LIN {X 0,Y 369.698,Z 75.747,A -85,B 0,C 180,E1 18351.289,E2 18351.289} C_VEL
LIN {X 0,Y 369.703,Z 75.746,A -85,B 0,C 180,E1 18347.187,E2 18347.187} C_VEL
LIN {X 0,Y 369.706,Z 75.742,A -85,B 0,C 180,E1 18343.18,E2 18343.18} C_VEL
LIN {X 0,Y 369.715,Z 75.74,A -85,B 0,C 180,E1 18339.085,E2 18339.085} C_VEL
LIN {X 0,Y 369.717,Z 75.741,A -85,B 0,C 180,E1 18335.047,E2 18335.047} C_VEL
LIN {X 0,Y 369.727,Z 75.74,A -85,B 0,C 180,E1 18330.868,E2 18330.868} C_VEL
LIN {X 0,Y 369.716,Z 75.743,A -85,B 0,C 180,E1 18326.888,E2 18326.888} C_VEL
LIN {X 0,Y 369.699,Z 75.747,A -85,B 0,C 180,E1 18322.713,E2 18322.713} C_VEL
LIN {X 0,Y 369.713,Z 75.939,A -85,B 0,C 180,E1 18320.54,E2 18320.54} C_VEL
LIN {X 0,Y 371.263,Z 79.57,A -85,B 0,C 180,E1 18319.328,E2 18319.328} C_VEL
LIN {X 0,Y 375.253,Z 88.261,A -85,B 0,C 180,E1 18316.782,E2 18316.782} C_VEL
LIN {X 0,Y 380.2,Z 100.385,A -85,B 0,C 180,E1 18313.761,E2 18313.761} C_VEL
LIN {X 0,Y 384.853,Z 112.745,A -85,B 0,C 180,E1 18311.095,E2 18311.095} C_VEL
LIN {X 0,Y 389.715,Z 127.844,A -85,B 0,C 180,E1 18308.272,E2 18308.272} C_VEL
LIN {X 0,Y 390.35,Z 131.11,A -85,B 0,C 180,E1 18307.748,E2 18307.748} C_VEL
LIN {X 0,Y 385.426,Z 162.448,A -85,B 0,C 180,E1 18304.176,E2 18304.176} C_VEL
LIN {X 0,Y 388.099,Z 187.157,A -85,B 0,C 180,E1 18303.373,E2 18303.373} C_VEL
LIN {X 0,Y 384.621,Z 335.093,A -85,B 0,C 180,E1 18300.587,E2 18300.587} C_VEL
LIN {X 0,Y 383.923,Z 357.134,A -85,B 0,C 180,E1 18300.105,E2 18300.105} C_VEL
LIN {X 0,Y 382.601,Z 375.427,A -85,B 0,C 180,E1 18299.449,E2 18299.449} C_VEL
LIN {X 0,Y 380.899,Z 392.959,A -85,B 0,C 180,E1 18298.539,E2 18298.539} C_VEL
LIN {X 0,Y 378.892,Z 410.258,A -85,B 0,C 180,E1 18297.334,E2 18297.334} C_VEL
LIN {X 0,Y 376.85,Z 426.215,A -85,B 0,C 180,E1 18295.917,E2 18295.917} C_VEL
LIN {X 0,Y 374.801,Z 441.299,A -85,B 0,C 180,E1 18294.258,E2 18294.258} C_VEL
LIN {X 0,Y 372.823,Z 455.891,A -85,B 0,C 180,E1 18292.295,E2 18292.295} C_VEL
LIN {X 0,Y 371.166,Z 468.894,A -85,B 0,C 180,E1 18290.171,E2 18290.171} C_VEL
LIN {X 0,Y 369.836,Z 480.915,A -85,B 0,C 180,E1 18287.789,E2 18287.789} C_VEL
LIN {X 0,Y 368.946,Z 491.438,A -85,B 0,C 180,E1 18285.242,E2 18285.242} C_VEL
LIN {X 0,Y 368.524,Z 500.454,A -85,B 0,C 180,E1 18282.537,E2 18282.537} C_VEL
LIN {X 0,Y 368.497,Z 507.488,A -85,B 0,C 180,E1 18279.844,E2 18279.844} C_VEL
LIN {X 0,Y 368.76,Z 512.975,A -85,B 0,C 180,E1 18277.009,E2 18277.009} C_VEL
LIN {X 0,Y 369.086,Z 516.444,A -85,B 0,C 180,E1 18274.351,E2 18274.351} C_VEL
LIN {X 0,Y 369.324,Z 518.28,A -85,B 0,C 180,E1 18271.708,E2 18271.708} C_VEL
LIN {X 0,Y 369.368,Z 518.495,A -85,B 0,C 180,E1 18269.071,E2 18269.071} C_VEL
LIN {X 0,Y 369.174,Z 517.092,A -85,B 0,C 180,E1 18266.43,E2 18266.43} C_VEL
LIN {X 0,Y 368.867,Z 514.053,A -85,B 0,C 180,E1 18263.777,E2 18263.777} C_VEL
LIN {X 0,Y 368.587,Z 509.317,A -85,B 0,C 180,E1 18261.106,E2 18261.106} C_VEL
LIN {X 0,Y 368.502,Z 502.683,A -85,B 0,C 180,E1 18258.379,E2 18258.379} C_VEL
LIN {X 0,Y 368.771,Z 494.305,A -85,B 0,C 180,E1 18255.717,E2 18255.717} C_VEL
LIN {X 0,Y 369.45,Z 484.245,A -85,B 0,C 180,E1 18253.169,E2 18253.169} C_VEL
LIN {X 0,Y 370.552,Z 472.63,A -85,B 0,C 180,E1 18250.782,E2 18250.782} C_VEL
LIN {X 0,Y 372.025,Z 459.458,A -85,B 0,C 180,E1 18248.562,E2 18248.562} C_VEL
LIN {X 0,Y 373.773,Z 445.023,A -85,B 0,C 180,E1 18246.569,E2 18246.569} C_VEL
LIN {X 0,Y 375.673,Z 429.361,A -85,B 0,C 180,E1 18244.811,E2 18244.811} C_VEL
LIN {X 0,Y 377.468,Z 413.842,A -85,B 0,C 180,E1 18243.408,E2 18243.408} C_VEL
LIN {X 0,Y 379.259,Z 396.749,A -85,B 0,C 180,E1 18242.186,E2 18242.186} C_VEL
LIN {X 0,Y 380.811,Z 379.266,A -85,B 0,C 180,E1 18241.242,E2 18241.242} C_VEL
LIN {X 0,Y 382.074,Z 360.639,A -85,B 0,C 180,E1 18240.542,E2 18240.542} C_VEL
LIN {X 0,Y 382.7,Z 340.596,A -85,B 0,C 180,E1 18240.083,E2 18240.083} C_VEL
LIN {X 0,Y 386.004,Z 174.055,A -85,B 0,C 180,E1 18237.005,E2 18237.005} C_VEL
LIN {X 0,Y 385.322,Z 157.356,A -85,B 0,C 180,E1 18236.581,E2 18236.581} C_VEL
LIN {X 0,Y 388.344,Z 121.359,A -85,B 0,C 180,E1 18234.252,E2 18234.252} C_VEL
LIN {X 0,Y 379.099,Z 97.949,A -85,B 0,C 180,E1 18231.701,E2 18231.701} C_VEL
LIN {X 0,Y 371.121,Z 79.333,A -85,B 0,C 180,E1 18229.442,E2 18229.442} C_VEL
LIN {X 0,Y 369.792,Z 76.095,A -85,B 0,C 180,E1 18228.97,E2 18228.97} C_VEL
LIN {X 0,Y 369.747,Z 75.737,A -85,B 0,C 180,E1 18228.095,E2 18228.095} C_VEL
LIN {X 0,Y 369.744,Z 75.737,A -85,B 0,C 180,E1 18224.005,E2 18224.005} C_VEL
LIN {X 0,Y 369.744,Z 75.744,A -85,B 0,C 180,E1 18219.829,E2 18219.829} C_VEL
LIN {X 0,Y 369.737,Z 75.735,A -85,B 0,C 180,E1 18215.74,E2 18215.74} C_VEL
LIN {X 0,Y 369.733,Z 75.734,A -85,B 0,C 180,E1 18211.591,E2 18211.591} C_VEL
LIN {X 0,Y 369.731,Z 75.733,A -85,B 0,C 180,E1 18207.505,E2 18207.505} C_VEL
LIN {X 0,Y 369.735,Z 75.729,A -85,B 0,C 180,E1 18203.423,E2 18203.423} C_VEL
LIN {X 0,Y 369.74,Z 75.73,A -85,B 0,C 180,E1 18199.311,E2 18199.311} C_VEL
LIN {X 0,Y 369.75,Z 75.733,A -85,B 0,C 180,E1 18195.129,E2 18195.129} C_VEL
LIN {X 0,Y 369.747,Z 75.739,A -85,B 0,C 180,E1 18191.015,E2 18191.015} C_VEL
LIN {X 0,Y 369.749,Z 75.742,A -85,B 0,C 180,E1 18186.833,E2 18186.833} C_VEL
LIN {X 0,Y 369.732,Z 75.743,A -85,B 0,C 180,E1 18182.635,E2 18182.635} C_VEL
LIN {X 0,Y 369.726,Z 75.738,A -85,B 0,C 180,E1 18178.605,E2 18178.605} C_VEL
LIN {X 0,Y 369.719,Z 75.734,A -85,B 0,C 180,E1 18174.568,E2 18174.568} C_VEL
LIN {X 0,Y 369.716,Z 75.732,A -85,B 0,C 180,E1 18170.504,E2 18170.504} C_VEL
LIN {X 0,Y 369.713,Z 75.733,A -85,B 0,C 180,E1 18166.391,E2 18166.391} C_VEL
LIN {X 0,Y 369.715,Z 75.735,A -85,B 0,C 180,E1 18162.368,E2 18162.368} C_VEL
LIN {X 0,Y 369.718,Z 75.729,A -85,B 0,C 180,E1 18158.253,E2 18158.253} C_VEL
LIN {X 0,Y 369.725,Z 75.734,A -85,B 0,C 180,E1 18154.189,E2 18154.189} C_VEL
LIN {X 0,Y 369.727,Z 75.716,A -85,B 0,C 180,E1 18150.159,E2 18150.159} C_VEL
LIN {X 0,Y 369.734,Z 75.739,A -85,B 0,C 180,E1 18146.117,E2 18146.117} C_VEL
LIN {X 0,Y 369.745,Z 75.747,A -85,B 0,C 180,E1 18141.895,E2 18141.895} C_VEL
LIN {X 0,Y 369.732,Z 75.746,A -85,B 0,C 180,E1 18137.811,E2 18137.811} C_VEL
LIN {X 0,Y 369.73,Z 75.854,A -85,B 0,C 180,E1 18133.661,E2 18133.661} C_VEL
LIN {X 0,Y 370.111,Z 77.451,A -85,B 0,C 180,E1 18133.326,E2 18133.326} C_VEL
LIN {X 0,Y 375.188,Z 90.914,A -85,B 0,C 180,E1 18131.164,E2 18131.164} C_VEL
LIN {X 0,Y 380.295,Z 107.557,A -85,B 0,C 180,E1 18128.66,E2 18128.66} C_VEL
LIN {X 0,Y 381.618,Z 113.58,A -85,B 0,C 180,E1 18127.811,E2 18127.811} C_VEL
LIN {X 0,Y 380.63,Z 148.33,A -85,B 0,C 180,E1 18123.749,E2 18123.749} C_VEL
LIN {X 0,Y 379.687,Z 184.035,A -85,B 0,C 180,E1 18119.655,E2 18119.655} C_VEL
LIN {X 0,Y 379.452,Z 200.957,A -85,B 0,C 180,E1 18117.821,E2 18117.821} C_VEL
LIN {X 0,Y 380.058,Z 205.985,A -85,B 0,C 180,E1 18117.673,E2 18117.673} C_VEL
LIN {X 0,Y 378.353,Z 307.859,A -85,B 0,C 180,E1 18115.716,E2 18115.716} C_VEL
LIN {X 0,Y 378.281,Z 322.743,A -85,B 0,C 180,E1 18115.252,E2 18115.252} C_VEL
LIN {X 0,Y 377.861,Z 336.788,A -85,B 0,C 180,E1 18114.545,E2 18114.545} C_VEL
LIN {X 0,Y 377.058,Z 350.975,A -85,B 0,C 180,E1 18113.519,E2 18113.519} C_VEL
LIN {X 0,Y 376.047,Z 363.63,A -85,B 0,C 180,E1 18112.287,E2 18112.287} C_VEL
LIN {X 0,Y 374.946,Z 375.143,A -85,B 0,C 180,E1 18110.836,E2 18110.836} C_VEL
LIN {X 0,Y 373.79,Z 385.284,A -85,B 0,C 180,E1 18109.207,E2 18109.207} C_VEL
LIN {X 0,Y 372.627,Z 394.373,A -85,B 0,C 180,E1 18107.327,E2 18107.327} C_VEL
LIN {X 0,Y 371.679,Z 401.417,A -85,B 0,C 180,E1 18105.444,E2 18105.444} C_VEL
LIN {X 0,Y 370.832,Z 407.525,A -85,B 0,C 180,E1 18103.247,E2 18103.247} C_VEL
LIN {X 0,Y 370.196,Z 411.9,A -85,B 0,C 180,E1 18100.897,E2 18100.897} C_VEL
LIN {X 0,Y 369.808,Z 414.328,A -85,B 0,C 180,E1 18098.551,E2 18098.551} C_VEL
LIN {X 0,Y 369.626,Z 414.959,A -85,B 0,C 180,E1 18096.21,E2 18096.21} C_VEL
LIN {X 0,Y 369.636,Z 413.831,A -85,B 0,C 180,E1 18093.876,E2 18093.876} C_VEL
LIN {X 0,Y 369.858,Z 410.615,A -85,B 0,C 180,E1 18091.393,E2 18091.393} C_VEL
LIN {X 0,Y 370.279,Z 405.57,A -85,B 0,C 180,E1 18089.071,E2 18089.071} C_VEL
LIN {X 0,Y 370.837,Z 399.392,A -85,B 0,C 180,E1 18087.062,E2 18087.062} C_VEL
LIN {X 0,Y 371.6,Z 391.246,A -85,B 0,C 180,E1 18085.06,E2 18085.06} C_VEL
LIN {X 0,Y 372.064,Z 386.159,A -85,B 0,C 180,E1 18084.043,E2 18084.043} C_VEL
LIN {X 0,Y 371.549,Z 381.232,A -85,B 0,C 180,E1 18083.121,E2 18083.121} C_VEL
LIN {X 0,Y 368.041,Z 371.768,A -85,B 0,C 180,E1 18081.5,E2 18081.5} C_VEL
LIN {X 0,Y 366.43,Z 365.291,A -85,B 0,C 180,E1 18080.582,E2 18080.582} C_VEL
LIN {X 0,Y 366.351,Z 361.699,A -85,B 0,C 180,E1 18080.163,E2 18080.163} C_VEL
LIN {X 0,Y 367.154,Z 348.44,A -85,B 0,C 180,E1 18078.93,E2 18078.93} C_VEL
LIN {X 0,Y 367.732,Z 334.792,A -85,B 0,C 180,E1 18077.994,E2 18077.994} C_VEL
LIN {X 0,Y 368,Z 320.348,A -85,B 0,C 180,E1 18077.305,E2 18077.305} C_VEL
LIN {X 0,Y 367.969,Z 303.735,A -85,B 0,C 180,E1 18076.855,E2 18076.855} C_VEL
LIN {X 0,Y 369.693,Z 197.834,A -85,B 0,C 180,E1 18074.79,E2 18074.79} C_VEL
LIN {X 0,Y 370.403,Z 188.265,A -85,B 0,C 180,E1 18074.178,E2 18074.178} C_VEL
LIN {X 0,Y 370.622,Z 185.191,A -85,B 0,C 180,E1 18073.906,E2 18073.906} C_VEL
LIN {X 0,Y 371.261,Z 184.243,A -85,B 0,C 180,E1 18073.653,E2 18073.653} C_VEL
LIN {X 0,Y 372.216,Z 184.586,A -85,B 0,C 180,E1 18073.476,E2 18073.476} C_VEL
LIN {X 0,Y 374.171,Z 186.02,A -85,B 0,C 180,E1 18073.295,E2 18073.295} C_VEL
LIN {X 0,Y 374.868,Z 197.394,A -85,B 0,C 180,E1 18072.973,E2 18072.973} C_VEL
LIN {X 0,Y 371.793,Z 301.218,A -85,B 0,C 180,E1 18070.645,E2 18070.645} C_VEL
LIN {X 0,Y 371.137,Z 317.525,A -85,B 0,C 180,E1 18069.992,E2 18069.992} C_VEL
LIN {X 0,Y 370.215,Z 332.434,A -85,B 0,C 180,E1 18069.114,E2 18069.114} C_VEL
LIN {X 0,Y 369.084,Z 346.795,A -85,B 0,C 180,E1 18067.986,E2 18067.986} C_VEL
LIN {X 0,Y 367.697,Z 361.204,A -85,B 0,C 180,E1 18066.5,E2 18066.5} C_VEL
LIN {X 0,Y 366.448,Z 373.045,A -85,B 0,C 180,E1 18064.941,E2 18064.941} C_VEL
LIN {X 0,Y 365.194,Z 383.994,A -85,B 0,C 180,E1 18063.143,E2 18063.143} C_VEL
LIN {X 0,Y 364.03,Z 393.789,A -85,B 0,C 180,E1 18061.091,E2 18061.091} C_VEL
LIN {X 0,Y 363.098,Z 401.859,A -85,B 0,C 180,E1 18058.915,E2 18058.915} C_VEL
LIN {X 0,Y 362.369,Z 408.627,A -85,B 0,C 180,E1 18056.439,E2 18056.439} C_VEL
LIN {X 0,Y 361.944,Z 413.075,A -85,B 0,C 180,E1 18054.039,E2 18054.039} C_VEL
LIN {X 0,Y 361.762,Z 415.798,A -85,B 0,C 180,E1 18051.547,E2 18051.547} C_VEL
LIN {X 0,Y 361.815,Z 416.609,A -85,B 0,C 180,E1 18048.976,E2 18048.976} C_VEL
LIN {X 0,Y 362.098,Z 415.605,A -85,B 0,C 180,E1 18046.562,E2 18046.562} C_VEL
LIN {X 0,Y 362.68,Z 412.568,A -85,B 0,C 180,E1 18043.983,E2 18043.983} C_VEL
LIN {X 0,Y 363.459,Z 408.133,A -85,B 0,C 180,E1 18041.739,E2 18041.739} C_VEL
LIN {X 0,Y 364.635,Z 401.413,A -85,B 0,C 180,E1 18039.351,E2 18039.351} C_VEL
LIN {X 0,Y 366.023,Z 393.164,A -85,B 0,C 180,E1 18037.196,E2 18037.196} C_VEL
LIN {X 0,Y 367.611,Z 383.402,A -85,B 0,C 180,E1 18035.213,E2 18035.213} C_VEL
LIN {X 0,Y 369.378,Z 371.52,A -85,B 0,C 180,E1 18033.333,E2 18033.333} C_VEL
LIN {X 0,Y 371.018,Z 359.359,A -85,B 0,C 180,E1 18031.817,E2 18031.817} C_VEL
LIN {X 0,Y 372.676,Z 345.086,A -85,B 0,C 180,E1 18030.42,E2 18030.42} C_VEL
LIN {X 0,Y 374.102,Z 329.6,A -85,B 0,C 180,E1 18029.282,E2 18029.282} C_VEL
LIN {X 0,Y 375.148,Z 314.19,A -85,B 0,C 180,E1 18028.461,E2 18028.461} C_VEL
LIN {X 0,Y 375.878,Z 297.331,A -85,B 0,C 180,E1 18027.87,E2 18027.87} C_VEL
LIN {X 0,Y 379.463,Z 207.466,A -85,B 0,C 180,E1 18025.682,E2 18025.682} C_VEL
LIN {X 0,Y 374.321,Z 178.027,A -85,B 0,C 180,E1 18024.332,E2 18024.332} C_VEL
LIN {X 0,Y 373.222,Z 172.209,A -85,B 0,C 180,E1 18024.001,E2 18024.001} C_VEL
LIN {X 0,Y 377.007,Z 145.712,A -85,B 0,C 180,E1 18019.683,E2 18019.683} C_VEL
LIN {X 0,Y 379.418,Z 130.52,A -85,B 0,C 180,E1 18017.167,E2 18017.167} C_VEL
LIN {X 0,Y 376.228,Z 117.259,A -85,B 0,C 180,E1 18014.153,E2 18014.153} C_VEL
LIN {X 0,Y 372.504,Z 104.805,A -85,B 0,C 180,E1 18010.987,E2 18010.987} C_VEL
LIN {X 0,Y 368.787,Z 94.247,A -85,B 0,C 180,E1 18007.948,E2 18007.948} C_VEL
LIN {X 0,Y 365.768,Z 86.709,A -85,B 0,C 180,E1 18005.491,E2 18005.491} C_VEL
LIN {X 0,Y 363.086,Z 80.246,A -85,B 0,C 180,E1 18003.158,E2 18003.158} C_VEL
LIN {X 0,Y 361.785,Z 76.834,A -85,B 0,C 180,E1 18001.742,E2 18001.742} C_VEL
LIN {X 0,Y 361.766,Z 76.732,A -85,B 0,C 180,E1 17997.783,E2 17997.783} C_VEL
LIN {X 0,Y 361.759,Z 76.733,A -85,B 0,C 180,E1 17993.653,E2 17993.653} C_VEL
LIN {X 0,Y 361.757,Z 76.734,A -85,B 0,C 180,E1 17989.49,E2 17989.49} C_VEL
LIN {X 0,Y 361.76,Z 76.732,A -85,B 0,C 180,E1 17985.321,E2 17985.321} C_VEL
LIN {X 0,Y 361.761,Z 76.73,A -85,B 0,C 180,E1 17981.301,E2 17981.301} C_VEL
LIN {X 0,Y 361.767,Z 76.73,A -85,B 0,C 180,E1 17977.236,E2 17977.236} C_VEL
LIN {X 0,Y 361.781,Z 76.729,A -85,B 0,C 180,E1 17973.048,E2 17973.048} C_VEL
LIN {X 0,Y 361.786,Z 76.73,A -85,B 0,C 180,E1 17968.882,E2 17968.882} C_VEL
LIN {X 0,Y 361.764,Z 76.738,A -85,B 0,C 180,E1 17964.715,E2 17964.715} C_VEL
LIN {X 0,Y 361.784,Z 77.027,A -85,B 0,C 180,E1 17962.286,E2 17962.286} C_VEL
LIN {X 0,Y 363.536,Z 80.865,A -85,B 0,C 180,E1 17960.861,E2 17960.861} C_VEL
LIN {X 0,Y 366.269,Z 87.098,A -85,B 0,C 180,E1 17958.861,E2 17958.861} C_VEL
LIN {X 0,Y 369.245,Z 93.448,A -85,B 0,C 180,E1 17956.971,E2 17956.971} C_VEL
LIN {X 0,Y 373.932,Z 105.09,A -85,B 0,C 180,E1 17954.005,E2 17954.005} C_VEL
LIN {X 0,Y 378.636,Z 117.95,A -85,B 0,C 180,E1 17951.185,E2 17951.185} C_VEL
LIN {X 0,Y 383.225,Z 132.648,A -85,B 0,C 180,E1 17948.387,E2 17948.387} C_VEL
LIN {X 0,Y 383.339,Z 133.981,A -85,B 0,C 180,E1 17948.183,E2 17948.183} C_VEL
LIN {X 0,Y 378.588,Z 162.637,A -85,B 0,C 180,E1 17944.852,E2 17944.852} C_VEL
LIN {X 0,Y 381.297,Z 187.979,A -85,B 0,C 180,E1 17943.991,E2 17943.991} C_VEL
LIN {X 0,Y 377.104,Z 352.179,A -85,B 0,C 180,E1 17940.807,E2 17940.807} C_VEL
LIN {X 0,Y 375.864,Z 370.525,A -85,B 0,C 180,E1 17940.195,E2 17940.195} C_VEL
LIN {X 0,Y 374.052,Z 388.976,A -85,B 0,C 180,E1 17939.287,E2 17939.287} C_VEL
LIN {X 0,Y 372.051,Z 406.054,A -85,B 0,C 180,E1 17938.142,E2 17938.142} C_VEL
LIN {X 0,Y 369.904,Z 422.137,A -85,B 0,C 180,E1 17936.76,E2 17936.76} C_VEL
LIN {X 0,Y 367.712,Z 437.614,A -85,B 0,C 180,E1 17935.1,E2 17935.1} C_VEL
LIN {X 0,Y 365.616,Z 452.083,A -85,B 0,C 180,E1 17933.192,E2 17933.192} C_VEL
LIN {X 0,Y 363.675,Z 465.993,A -85,B 0,C 180,E1 17930.942,E2 17930.942} C_VEL
LIN {X 0,Y 362.166,Z 478.323,A -85,B 0,C 180,E1 17928.512,E2 17928.512} C_VEL
LIN {X 0,Y 361.12,Z 489.113,A -85,B 0,C 180,E1 17925.91,E2 17925.91} C_VEL
LIN {X 0,Y 360.586,Z 498.36,A -85,B 0,C 180,E1 17923.144,E2 17923.144} C_VEL
LIN {X 0,Y 360.493,Z 505.612,A -85,B 0,C 180,E1 17920.387,E2 17920.387} C_VEL
LIN {X 0,Y 360.724,Z 511.064,A -85,B 0,C 180,E1 17917.647,E2 17917.647} C_VEL
LIN {X 0,Y 361.07,Z 514.813,A -85,B 0,C 180,E1 17914.926,E2 17914.926} C_VEL
LIN {X 0,Y 361.364,Z 516.927,A -85,B 0,C 180,E1 17912.221,E2 17912.221} C_VEL
LIN {X 0,Y 361.457,Z 517.425,A -85,B 0,C 180,E1 17909.526,E2 17909.526} C_VEL
LIN {X 0,Y 361.286,Z 516.294,A -85,B 0,C 180,E1 17906.828,E2 17906.828} C_VEL
LIN {X 0,Y 360.963,Z 513.519,A -85,B 0,C 180,E1 17904.119,E2 17904.119} C_VEL
LIN {X 0,Y 360.649,Z 509.047,A -85,B 0,C 180,E1 17901.391,E2 17901.391} C_VEL
LIN {X 0,Y 360.519,Z 502.362,A -85,B 0,C 180,E1 17898.483,E2 17898.483} C_VEL
LIN {X 0,Y 360.748,Z 494.584,A -85,B 0,C 180,E1 17895.884,E2 17895.884} C_VEL
LIN {X 0,Y 361.398,Z 484.846,A -85,B 0,C 180,E1 17893.279,E2 17893.279} C_VEL
LIN {X 0,Y 362.492,Z 473.616,A -85,B 0,C 180,E1 17890.84,E2 17890.84} C_VEL
LIN {X 0,Y 363.968,Z 460.882,A -85,B 0,C 180,E1 17888.572,E2 17888.572} C_VEL
LIN {X 0,Y 365.777,Z 446.469,A -85,B 0,C 180,E1 17886.48,E2 17886.48} C_VEL
LIN {X 0,Y 367.66,Z 431.673,A -85,B 0,C 180,E1 17884.727,E2 17884.727} C_VEL
LIN {X 0,Y 369.57,Z 416.07,A -85,B 0,C 180,E1 17883.227,E2 17883.227} C_VEL
LIN {X 0,Y 371.385,Z 399.763,A -85,B 0,C 180,E1 17881.981,E2 17881.981} C_VEL
LIN {X 0,Y 373.104,Z 381.924,A -85,B 0,C 180,E1 17880.942,E2 17880.942} C_VEL
LIN {X 0,Y 374.476,Z 363.631,A -85,B 0,C 180,E1 17880.185,E2 17880.185} C_VEL
LIN {X 0,Y 375.234,Z 345.261,A -85,B 0,C 180,E1 17879.701,E2 17879.701} C_VEL
LIN {X 0,Y 378.813,Z 174.715,A -85,B 0,C 180,E1 17876.489,E2 17876.489} C_VEL
LIN {X 0,Y 378.136,Z 157.313,A -85,B 0,C 180,E1 17876.036,E2 17876.036} C_VEL
LIN {X 0,Y 381.061,Z 123.76,A -85,B 0,C 180,E1 17873.819,E2 17873.819} C_VEL
LIN {X 0,Y 371.694,Z 99.975,A -85,B 0,C 180,E1 17871.147,E2 17871.147} C_VEL
LIN {X 0,Y 362.82,Z 79.739,A -85,B 0,C 180,E1 17868.596,E2 17868.596} C_VEL
LIN {X 0,Y 361.856,Z 77.053,A -85,B 0,C 180,E1 17868.192,E2 17868.192} C_VEL
LIN {X 0,Y 361.8,Z 76.732,A -85,B 0,C 180,E1 17867.172,E2 17867.172} C_VEL
LIN {X 0,Y 361.804,Z 76.729,A -85,B 0,C 180,E1 17862.92,E2 17862.92} C_VEL
LIN {X 0,Y 361.813,Z 76.725,A -85,B 0,C 180,E1 17858.807,E2 17858.807} C_VEL
LIN {X 0,Y 361.81,Z 76.723,A -85,B 0,C 180,E1 17854.565,E2 17854.565} C_VEL
LIN {X 0,Y 361.815,Z 76.727,A -85,B 0,C 180,E1 17850.378,E2 17850.378} C_VEL
LIN {X 0,Y 361.803,Z 76.729,A -85,B 0,C 180,E1 17846.242,E2 17846.242} C_VEL
LIN {X 0,Y 361.797,Z 76.729,A -85,B 0,C 180,E1 17842.076,E2 17842.076} C_VEL
LIN {X 0,Y 361.788,Z 76.728,A -85,B 0,C 180,E1 17837.864,E2 17837.864} C_VEL
LIN {X 0,Y 361.788,Z 76.722,A -85,B 0,C 180,E1 17833.749,E2 17833.749} C_VEL
LIN {X 0,Y 361.794,Z 76.716,A -85,B 0,C 180,E1 17829.544,E2 17829.544} C_VEL
LIN {X 0,Y 361.797,Z 76.724,A -85,B 0,C 180,E1 17825.55,E2 17825.55} C_VEL
LIN {X 0,Y 361.805,Z 76.728,A -85,B 0,C 180,E1 17821.425,E2 17821.425} C_VEL
LIN {X 0,Y 361.806,Z 76.73,A -85,B 0,C 180,E1 17817.307,E2 17817.307} C_VEL
LIN {X 0,Y 361.813,Z 76.728,A -85,B 0,C 180,E1 17813.175,E2 17813.175} C_VEL
LIN {X 0,Y 361.793,Z 76.728,A -85,B 0,C 180,E1 17809.007,E2 17809.007} C_VEL
LIN {X 0,Y 361.785,Z 76.727,A -85,B 0,C 180,E1 17804.942,E2 17804.942} C_VEL
LIN {X 0,Y 361.777,Z 76.731,A -85,B 0,C 180,E1 17800.798,E2 17800.798} C_VEL
LIN {X 0,Y 361.772,Z 76.694,A -85,B 0,C 180,E1 17796.547,E2 17796.547} C_VEL
LIN {X 0,Y 361.775,Z 76.733,A -85,B 0,C 180,E1 17792.512,E2 17792.512} C_VEL
LIN {X 0,Y 361.773,Z 76.716,A -85,B 0,C 180,E1 17788.509,E2 17788.509} C_VEL
LIN {X 0,Y 361.772,Z 76.712,A -85,B 0,C 180,E1 17784.521,E2 17784.521} C_VEL
LIN {X 0,Y 361.778,Z 76.72,A -85,B 0,C 180,E1 17780.448,E2 17780.448} C_VEL
LIN {X 0,Y 361.791,Z 76.718,A -85,B 0,C 180,E1 17776.297,E2 17776.297} C_VEL
LIN {X 0,Y 361.825,Z 76.996,A -85,B 0,C 180,E1 17774.382,E2 17774.382} C_VEL
LIN {X 0,Y 368.457,Z 95.021,A -85,B 0,C 180,E1 17771.381,E2 17771.381} C_VEL
LIN {X 0,Y 373.513,Z 111.76,A -85,B 0,C 180,E1 17768.832,E2 17768.832} C_VEL
LIN {X 0,Y 374.46,Z 116.271,A -85,B 0,C 180,E1 17768.188,E2 17768.188} C_VEL
LIN {X 0,Y 373.374,Z 151.557,A -85,B 0,C 180,E1 17764.032,E2 17764.032} C_VEL
LIN {X 0,Y 372.387,Z 187.837,A -85,B 0,C 180,E1 17759.858,E2 17759.858} C_VEL
LIN {X 0,Y 372.146,Z 201.909,A -85,B 0,C 180,E1 17758.325,E2 17758.325} C_VEL
LIN {X 0,Y 372.787,Z 207.087,A -85,B 0,C 180,E1 17758.168,E2 17758.168} C_VEL
LIN {X 0,Y 370.982,Z 308.241,A -85,B 0,C 180,E1 17756.189,E2 17756.189} C_VEL
LIN {X 0,Y 370.914,Z 323.342,A -85,B 0,C 180,E1 17755.72,E2 17755.72} C_VEL
LIN {X 0,Y 370.457,Z 337.796,A -85,B 0,C 180,E1 17754.984,E2 17754.984} C_VEL
LIN {X 0,Y 369.609,Z 352.011,A -85,B 0,C 180,E1 17753.938,E2 17753.938} C_VEL
LIN {X 0,Y 368.582,Z 364.251,A -85,B 0,C 180,E1 17752.731,E2 17752.731} C_VEL
LIN {X 0,Y 367.455,Z 375.561,A -85,B 0,C 180,E1 17751.299,E2 17751.299} C_VEL
LIN {X 0,Y 366.099,Z 386.791,A -85,B 0,C 180,E1 17749.461,E2 17749.461} C_VEL
LIN {X 0,Y 364.786,Z 396.461,A -85,B 0,C 180,E1 17747.382,E2 17747.382} C_VEL
LIN {X 0,Y 363.658,Z 404.236,A -85,B 0,C 180,E1 17745.14,E2 17745.14} C_VEL
LIN {X 0,Y 362.814,Z 409.801,A -85,B 0,C 180,E1 17742.897,E2 17742.897} C_VEL
LIN {X 0,Y 362.233,Z 413.52,A -85,B 0,C 180,E1 17740.656,E2 17740.656} C_VEL
LIN {X 0,Y 361.855,Z 415.673,A -85,B 0,C 180,E1 17738.26,E2 17738.26} C_VEL
LIN {X 0,Y 361.688,Z 415.965,A -85,B 0,C 180,E1 17735.71,E2 17735.71} C_VEL
LIN {X 0,Y 361.747,Z 414.228,A -85,B 0,C 180,E1 17733.168,E2 17733.168} C_VEL
LIN {X 0,Y 362.019,Z 410.7,A -85,B 0,C 180,E1 17730.79,E2 17730.79} C_VEL
LIN {X 0,Y 362.475,Z 405.614,A -85,B 0,C 180,E1 17728.576,E2 17728.576} C_VEL
LIN {X 0,Y 363.106,Z 399.118,A -85,B 0,C 180,E1 17726.526,E2 17726.526} C_VEL
LIN {X 0,Y 363.944,Z 390.508,A -85,B 0,C 180,E1 17724.481,E2 17724.481} C_VEL
LIN {X 0,Y 364.816,Z 381.152,A -85,B 0,C 180,E1 17722.756,E2 17722.756} C_VEL
LIN {X 0,Y 365.775,Z 369.814,A -85,B 0,C 180,E1 17721.114,E2 17721.114} C_VEL
LIN {X 0,Y 366.351,Z 361.699,A -85,B 0,C 180,E1 17720.163,E2 17720.163} C_VEL
LIN {X 0,Y 365.835,Z 355.352,A -85,B 0,C 180,E1 17719.464,E2 17719.464} C_VEL
LIN {X 0,Y 362.537,Z 344.434,A -85,B 0,C 180,E1 17718.347,E2 17718.347} C_VEL
LIN {X 0,Y 360.593,Z 336.68,A -85,B 0,C 180,E1 17717.72,E2 17717.72} C_VEL
LIN {X 0,Y 360.219,Z 331.508,A -85,B 0,C 180,E1 17717.407,E2 17717.407} C_VEL
LIN {X 0,Y 360.411,Z 316.564,A -85,B 0,C 180,E1 17716.778,E2 17716.778} C_VEL
LIN {X 0,Y 360.589,Z 278.756,A -85,B 0,C 180,E1 17715.965,E2 17715.965} C_VEL
LIN {X 0,Y 362.164,Z 199.347,A -85,B 0,C 180,E1 17714.384,E2 17714.384} C_VEL
LIN {X 0,Y 362.67,Z 196.935,A -85,B 0,C 180,E1 17714.16,E2 17714.16} C_VEL
LIN {X 0,Y 363.659,Z 196.064,A -85,B 0,C 180,E1 17713.876,E2 17713.876} C_VEL
LIN {X 0,Y 365.776,Z 197.599,A -85,B 0,C 180,E1 17713.633,E2 17713.633} C_VEL
LIN {X 0,Y 367.619,Z 197.786,A -85,B 0,C 180,E1 17713.492,E2 17713.492} C_VEL
LIN {X 0,Y 364.392,Z 301.648,A -85,B 0,C 180,E1 17711.113,E2 17711.113} C_VEL
LIN {X 0,Y 363.702,Z 318.046,A -85,B 0,C 180,E1 17710.445,E2 17710.445} C_VEL
LIN {X 0,Y 362.69,Z 333.639,A -85,B 0,C 180,E1 17709.505,E2 17709.505} C_VEL
LIN {X 0,Y 361.488,Z 348.073,A -85,B 0,C 180,E1 17708.337,E2 17708.337} C_VEL
LIN {X 0,Y 360.041,Z 362.488,A -85,B 0,C 180,E1 17706.812,E2 17706.812} C_VEL
LIN {X 0,Y 358.642,Z 375.026,A -85,B 0,C 180,E1 17705.103,E2 17705.103} C_VEL
LIN {X 0,Y 357.319,Z 385.995,A -85,B 0,C 180,E1 17703.222,E2 17703.222} C_VEL
LIN {X 0,Y 356.128,Z 395.608,A -85,B 0,C 180,E1 17701.124,E2 17701.124} C_VEL
LIN {X 0,Y 355.204,Z 403.19,A -85,B 0,C 180,E1 17698.993,E2 17698.993} C_VEL
LIN {X 0,Y 354.484,Z 409.569,A -85,B 0,C 180,E1 17696.606,E2 17696.606} C_VEL
LIN {X 0,Y 354.044,Z 413.975,A -85,B 0,C 180,E1 17694.225,E2 17694.225} C_VEL
LIN {X 0,Y 353.844,Z 416.737,A -85,B 0,C 180,E1 17691.769,E2 17691.769} C_VEL
LIN {X 0,Y 353.877,Z 417.734,A -85,B 0,C 180,E1 17689.22,E2 17689.22} C_VEL
LIN {X 0,Y 354.167,Z 416.947,A -85,B 0,C 180,E1 17686.683,E2 17686.683} C_VEL
LIN {X 0,Y 354.697,Z 414.42,A -85,B 0,C 180,E1 17684.274,E2 17684.274} C_VEL
LIN {X 0,Y 355.553,Z 410.005,A -85,B 0,C 180,E1 17681.796,E2 17681.796} C_VEL
LIN {X 0,Y 356.659,Z 404.042,A -85,B 0,C 180,E1 17679.522,E2 17679.522} C_VEL
LIN {X 0,Y 358.106,Z 396.168,A -85,B 0,C 180,E1 17677.274,E2 17677.274} C_VEL
LIN {X 0,Y 359.759,Z 386.663,A -85,B 0,C 180,E1 17675.204,E2 17675.204} C_VEL
LIN {X 0,Y 361.517,Z 375.933,A -85,B 0,C 180,E1 17673.357,E2 17673.357} C_VEL
LIN {X 0,Y 363.433,Z 362.862,A -85,B 0,C 180,E1 17671.599,E2 17671.599} C_VEL
LIN {X 0,Y 365.04,Z 350.233,A -85,B 0,C 180,E1 17670.264,E2 17670.264} C_VEL
LIN {X 0,Y 366.612,Z 335.35,A -85,B 0,C 180,E1 17669.043,E2 17669.043} C_VEL
LIN {X 0,Y 367.802,Z 320.518,A -85,B 0,C 180,E1 17668.142,E2 17668.142} C_VEL
LIN {X 0,Y 368.713,Z 304.032,A -85,B 0,C 180,E1 17667.447,E2 17667.447} C_VEL
LIN {X 0,Y 372.74,Z 208.847,A -85,B 0,C 180,E1 17665.045,E2 17665.045} C_VEL
LIN {X 0,Y 367.735,Z 179.907,A -85,B 0,C 180,E1 17663.676,E2 17663.676} C_VEL
LIN {X 0,Y 366.264,Z 172.119,A -85,B 0,C 180,E1 17663.233,E2 17663.233} C_VEL
LIN {X 0,Y 370.459,Z 144.692,A -85,B 0,C 180,E1 17658.676,E2 17658.676} C_VEL
LIN {X 0,Y 372.276,Z 133.118,A -85,B 0,C 180,E1 17656.702,E2 17656.702} C_VEL
LIN {X 0,Y 369.147,Z 120.062,A -85,B 0,C 180,E1 17653.63,E2 17653.63} C_VEL
LIN {X 0,Y 365.502,Z 107.842,A -85,B 0,C 180,E1 17650.402,E2 17650.402} C_VEL
LIN {X 0,Y 361.732,Z 96.884,A -85,B 0,C 180,E1 17647.11,E2 17647.11} C_VEL
LIN {X 0,Y 358.264,Z 88.443,A -85,B 0,C 180,E1 17644.161,E2 17644.161} C_VEL
LIN {X 0,Y 356.657,Z 84.754,A -85,B 0,C 180,E1 17642.732,E2 17642.732} C_VEL
LIN {X 0,Y 355.168,Z 81.263,A -85,B 0,C 180,E1 17641.291,E2 17641.291} C_VEL
LIN {X 0,Y 353.84,Z 77.821,A -85,B 0,C 180,E1 17639.677,E2 17639.677} C_VEL
LIN {X 0,Y 353.821,Z 77.723,A -85,B 0,C 180,E1 17635.462,E2 17635.462} C_VEL
LIN {X 0,Y 353.819,Z 77.724,A -85,B 0,C 180,E1 17631.387,E2 17631.387} C_VEL
LIN {X 0,Y 353.822,Z 77.723,A -85,B 0,C 180,E1 17627.267,E2 17627.267} C_VEL
LIN {X 0,Y 353.824,Z 77.719,A -85,B 0,C 180,E1 17623.248,E2 17623.248} C_VEL
LIN {X 0,Y 353.833,Z 77.718,A -85,B 0,C 180,E1 17619.142,E2 17619.142} C_VEL
LIN {X 0,Y 353.837,Z 77.719,A -85,B 0,C 180,E1 17615.1,E2 17615.1} C_VEL
LIN {X 0,Y 353.85,Z 77.717,A -85,B 0,C 180,E1 17610.921,E2 17610.921} C_VEL
LIN {X 0,Y 353.83,Z 77.723,A -85,B 0,C 180,E1 17606.756,E2 17606.756} C_VEL
LIN {X 0,Y 353.847,Z 78.002,A -85,B 0,C 180,E1 17604.357,E2 17604.357} C_VEL
LIN {X 0,Y 355.608,Z 81.866,A -85,B 0,C 180,E1 17602.723,E2 17602.723} C_VEL
LIN {X 0,Y 358.394,Z 87.994,A -85,B 0,C 180,E1 17600.5,E2 17600.5} C_VEL
LIN {X 0,Y 360.346,Z 92.27,A -85,B 0,C 180,E1 17599.093,E2 17599.093} C_VEL
LIN {X 0,Y 363.451,Z 99.3,A -85,B 0,C 180,E1 17596.98,E2 17596.98} C_VEL
LIN {X 0,Y 367.851,Z 110.259,A -85,B 0,C 180,E1 17594.145,E2 17594.145} C_VEL
LIN {X 0,Y 372.277,Z 122.757,A -85,B 0,C 180,E1 17591.354,E2 17591.354} C_VEL
LIN {X 0,Y 376.447,Z 136.342,A -85,B 0,C 180,E1 17588.71,E2 17588.71} C_VEL
LIN {X 0,Y 371.797,Z 162.756,A -85,B 0,C 180,E1 17585.557,E2 17585.557} C_VEL
LIN {X 0,Y 374.58,Z 188.805,A -85,B 0,C 180,E1 17584.642,E2 17584.642} C_VEL
LIN {X 0,Y 370.755,Z 330.501,A -85,B 0,C 180,E1 17581.863,E2 17581.863} C_VEL
LIN {X 0,Y 369.948,Z 355.039,A -85,B 0,C 180,E1 17581.322,E2 17581.322} C_VEL
LIN {X 0,Y 368.544,Z 373.254,A -85,B 0,C 180,E1 17580.656,E2 17580.656} C_VEL
LIN {X 0,Y 366.706,Z 390.409,A -85,B 0,C 180,E1 17579.752,E2 17579.752} C_VEL
LIN {X 0,Y 364.628,Z 406.941,A -85,B 0,C 180,E1 17578.588,E2 17578.588} C_VEL
LIN {X 0,Y 362.256,Z 423.509,A -85,B 0,C 180,E1 17577.092,E2 17577.092} C_VEL
LIN {X 0,Y 359.898,Z 439.072,A -85,B 0,C 180,E1 17575.331,E2 17575.331} C_VEL
LIN {X 0,Y 357.659,Z 453.627,A -85,B 0,C 180,E1 17573.303,E2 17573.303} C_VEL
LIN {X 0,Y 355.727,Z 466.784,A -85,B 0,C 180,E1 17571.066,E2 17571.066} C_VEL
LIN {X 0,Y 354.19,Z 478.696,A -85,B 0,C 180,E1 17568.603,E2 17568.603} C_VEL
LIN {X 0,Y 353.12,Z 489.231,A -85,B 0,C 180,E1 17565.942,E2 17565.942} C_VEL
LIN {X 0,Y 352.586,Z 498.251,A -85,B 0,C 180,E1 17563.113,E2 17563.113} C_VEL
LIN {X 0,Y 352.52,Z 505.62,A -85,B 0,C 180,E1 17560.129,E2 17560.129} C_VEL
LIN {X 0,Y 352.801,Z 510.818,A -85,B 0,C 180,E1 17557.29,E2 17557.29} C_VEL
LIN {X 0,Y 353.174,Z 514.23,A -85,B 0,C 180,E1 17554.548,E2 17554.548} C_VEL
LIN {X 0,Y 353.464,Z 516.065,A -85,B 0,C 180,E1 17551.784,E2 17551.784} C_VEL
LIN {X 0,Y 353.52,Z 516.258,A -85,B 0,C 180,E1 17549.029,E2 17549.029} C_VEL
LIN {X 0,Y 353.292,Z 514.803,A -85,B 0,C 180,E1 17546.269,E2 17546.269} C_VEL
LIN {X 0,Y 352.936,Z 511.691,A -85,B 0,C 180,E1 17543.495,E2 17543.495} C_VEL
LIN {X 0,Y 352.617,Z 506.801,A -85,B 0,C 180,E1 17540.667,E2 17540.667} C_VEL
LIN {X 0,Y 352.562,Z 499.782,A -85,B 0,C 180,E1 17537.721,E2 17537.721} C_VEL
LIN {X 0,Y 352.904,Z 491.513,A -85,B 0,C 180,E1 17535.045,E2 17535.045} C_VEL
LIN {X 0,Y 353.723,Z 481.287,A -85,B 0,C 180,E1 17532.397,E2 17532.397} C_VEL
LIN {X 0,Y 354.998,Z 469.446,A -85,B 0,C 180,E1 17529.904,E2 17529.904} C_VEL
LIN {X 0,Y 356.69,Z 455.998,A -85,B 0,C 180,E1 17527.592,E2 17527.592} C_VEL
LIN {X 0,Y 358.555,Z 442.045,A -85,B 0,C 180,E1 17525.627,E2 17525.627} C_VEL
LIN {X 0,Y 360.618,Z 426.52,A -85,B 0,C 180,E1 17523.844,E2 17523.844} C_VEL
LIN {X 0,Y 362.642,Z 410.334,A -85,B 0,C 180,E1 17522.355,E2 17522.355} C_VEL
LIN {X 0,Y 364.538,Z 393.371,A -85,B 0,C 180,E1 17521.138,E2 17521.138} C_VEL
LIN {X 0,Y 366.196,Z 375.476,A -85,B 0,C 180,E1 17520.182,E2 17520.182} C_VEL
LIN {X 0,Y 367.443,Z 357.252,A -85,B 0,C 180,E1 17519.511,E2 17519.511} C_VEL
LIN {X 0,Y 368.127,Z 333.318,A -85,B 0,C 180,E1 17518.985,E2 17518.985} C_VEL
LIN {X 0,Y 371.628,Z 174.883,A -85,B 0,C 180,E1 17515.94,E2 17515.94} C_VEL
LIN {X 0,Y 370.985,Z 157.281,A -85,B 0,C 180,E1 17515.471,E2 17515.471} C_VEL
LIN {X 0,Y 373.851,Z 126.327,A -85,B 0,C 180,E1 17513.389,E2 17513.389} C_VEL
LIN {X 0,Y 364.286,Z 102.081,A -85,B 0,C 180,E1 17510.591,E2 17510.591} C_VEL
LIN {X 0,Y 355.483,Z 81.7,A -85,B 0,C 180,E1 17507.948,E2 17507.948} C_VEL
LIN {X 0,Y 353.927,Z 78.148,A -85,B 0,C 180,E1 17507.412,E2 17507.412} C_VEL
LIN {X 0,Y 353.865,Z 77.72,A -85,B 0,C 180,E1 17506.863,E2 17506.863} C_VEL
LIN {X 0,Y 353.869,Z 77.719,A -85,B 0,C 180,E1 17502.697,E2 17502.697} C_VEL
LIN {X 0,Y 353.872,Z 77.712,A -85,B 0,C 180,E1 17498.499,E2 17498.499} C_VEL
LIN {X 0,Y 353.867,Z 77.715,A -85,B 0,C 180,E1 17494.213,E2 17494.213} C_VEL
LIN {X 0,Y 353.865,Z 77.721,A -85,B 0,C 180,E1 17490.008,E2 17490.008} C_VEL
LIN {X 0,Y 353.854,Z 77.72,A -85,B 0,C 180,E1 17485.794,E2 17485.794} C_VEL
LIN {X 0,Y 353.855,Z 77.719,A -85,B 0,C 180,E1 17481.551,E2 17481.551} C_VEL
LIN {X 0,Y 353.857,Z 77.717,A -85,B 0,C 180,E1 17477.428,E2 17477.428} C_VEL
LIN {X 0,Y 353.87,Z 77.71,A -85,B 0,C 180,E1 17473.23,E2 17473.23} C_VEL
LIN {X 0,Y 353.869,Z 77.705,A -85,B 0,C 180,E1 17468.94,E2 17468.94} C_VEL
LIN {X 0,Y 353.863,Z 77.705,A -85,B 0,C 180,E1 17464.862,E2 17464.862} C_VEL
LIN {X 0,Y 353.852,Z 77.708,A -85,B 0,C 180,E1 17460.647,E2 17460.647} C_VEL
LIN {X 0,Y 353.843,Z 77.716,A -85,B 0,C 180,E1 17456.436,E2 17456.436} C_VEL
LIN {X 0,Y 353.84,Z 77.72,A -85,B 0,C 180,E1 17452.204,E2 17452.204} C_VEL
LIN {X 0,Y 353.843,Z 77.72,A -85,B 0,C 180,E1 17448.095,E2 17448.095} C_VEL
LIN {X 0,Y 353.854,Z 77.719,A -85,B 0,C 180,E1 17443.924,E2 17443.924} C_VEL
LIN {X 0,Y 353.867,Z 77.72,A -85,B 0,C 180,E1 17439.663,E2 17439.663} C_VEL
LIN {X 0,Y 353.854,Z 77.684,A -85,B 0,C 180,E1 17435.457,E2 17435.457} C_VEL
LIN {X 0,Y 353.843,Z 77.706,A -85,B 0,C 180,E1 17431.29,E2 17431.29} C_VEL
LIN {X 0,Y 353.833,Z 77.726,A -85,B 0,C 180,E1 17427.142,E2 17427.142} C_VEL
LIN {X 0,Y 353.828,Z 77.713,A -85,B 0,C 180,E1 17422.993,E2 17422.993} C_VEL
LIN {X 0,Y 353.83,Z 77.712,A -85,B 0,C 180,E1 17418.732,E2 17418.732} C_VEL
LIN {X 0,Y 353.843,Z 77.854,A -85,B 0,C 180,E1 17415.283,E2 17415.283} C_VEL
LIN {X 0,Y 354.458,Z 79.983,A -85,B 0,C 180,E1 17414.843,E2 17414.843} C_VEL
LIN {X 0,Y 359.724,Z 93.329,A -85,B 0,C 180,E1 17412.559,E2 17412.559} C_VEL
LIN {X 0,Y 365.083,Z 109.949,A -85,B 0,C 180,E1 17409.928,E2 17409.928} C_VEL
LIN {X 0,Y 367.319,Z 119.159,A -85,B 0,C 180,E1 17408.559,E2 17408.559} C_VEL
LIN {X 0,Y 366.221,Z 152.529,A -85,B 0,C 180,E1 17404.601,E2 17404.601} C_VEL
LIN {X 0,Y 365.151,Z 188.816,A -85,B 0,C 180,E1 17400.397,E2 17400.397} C_VEL
LIN {X 0,Y 364.907,Z 203.039,A -85,B 0,C 180,E1 17398.844,E2 17398.844} C_VEL
LIN {X 0,Y 365.543,Z 208.362,A -85,B 0,C 180,E1 17398.681,E2 17398.681} C_VEL
LIN {X 0,Y 363.638,Z 308.601,A -85,B 0,C 180,E1 17396.681,E2 17396.681} C_VEL
LIN {X 0,Y 363.573,Z 323.955,A -85,B 0,C 180,E1 17396.207,E2 17396.207} C_VEL
LIN {X 0,Y 363.078,Z 338.814,A -85,B 0,C 180,E1 17395.44,E2 17395.44} C_VEL
LIN {X 0,Y 362.204,Z 352.748,A -85,B 0,C 180,E1 17394.4,E2 17394.4} C_VEL
LIN {X 0,Y 361.106,Z 365.24,A -85,B 0,C 180,E1 17393.151,E2 17393.151} C_VEL
LIN {X 0,Y 359.907,Z 376.631,A -85,B 0,C 180,E1 17391.682,E2 17391.682} C_VEL
LIN {X 0,Y 358.532,Z 387.432,A -85,B 0,C 180,E1 17389.889,E2 17389.889} C_VEL
LIN {X 0,Y 357.188,Z 396.783,A -85,B 0,C 180,E1 17387.87,E2 17387.87} C_VEL
LIN {X 0,Y 356.069,Z 404.084,A -85,B 0,C 180,E1 17385.804,E2 17385.804} C_VEL
LIN {X 0,Y 355.121,Z 410.048,A -85,B 0,C 180,E1 17383.513,E2 17383.513} C_VEL
LIN {X 0,Y 354.413,Z 414.316,A -85,B 0,C 180,E1 17381.059,E2 17381.059} C_VEL
LIN {X 0,Y 353.957,Z 416.726,A -85,B 0,C 180,E1 17378.445,E2 17378.445} C_VEL
LIN {X 0,Y 353.763,Z 417.074,A -85,B 0,C 180,E1 17375.839,E2 17375.839} C_VEL
LIN {X 0,Y 353.802,Z 415.559,A -85,B 0,C 180,E1 17373.401,E2 17373.401} C_VEL
LIN {X 0,Y 354.041,Z 412.53,A -85,B 0,C 180,E1 17371.132,E2 17371.132} C_VEL
LIN {X 0,Y 354.524,Z 407.371,A -85,B 0,C 180,E1 17368.706,E2 17368.706} C_VEL
LIN {X 0,Y 355.213,Z 400.495,A -85,B 0,C 180,E1 17366.448,E2 17366.448} C_VEL
LIN {X 0,Y 356.008,Z 392.716,A -85,B 0,C 180,E1 17364.519,E2 17364.519} C_VEL
LIN {X 0,Y 356.907,Z 383.692,A -85,B 0,C 180,E1 17362.757,E2 17362.757} C_VEL
LIN {X 0,Y 357.943,Z 372.129,A -85,B 0,C 180,E1 17360.999,E2 17360.999} C_VEL
LIN {X 0,Y 358.839,Z 359.906,A -85,B 0,C 180,E1 17359.564,E2 17359.564} C_VEL
LIN {X 0,Y 359.594,Z 347.574,A -85,B 0,C 180,E1 17358.45,E2 17358.45} C_VEL
LIN {X 0,Y 360.182,Z 333.172,A -85,B 0,C 180,E1 17357.494,E2 17357.494} C_VEL
LIN {X 0,Y 360.219,Z 331.508,A -85,B 0,C 180,E1 17357.407,E2 17357.407} C_VEL
LIN {X 0,Y 359.5,Z 324.174,A -85,B 0,C 180,E1 17357.012,E2 17357.012} C_VEL
LIN {X 0,Y 355.672,Z 311.9,A -85,B 0,C 180,E1 17356.396,E2 17356.396} C_VEL
LIN {X 0,Y 353.119,Z 302.437,A -85,B 0,C 180,E1 17356.053,E2 17356.053} C_VEL
LIN {X 0,Y 352.754,Z 298.07,A -85,B 0,C 180,E1 17355.943,E2 17355.943} C_VEL
LIN {X 0,Y 354.232,Z 221.304,A -85,B 0,C 180,E1 17354.361,E2 17354.361} C_VEL
LIN {X 0,Y 354.791,Z 218.134,A -85,B 0,C 180,E1 17354.135,E2 17354.135} C_VEL
LIN {X 0,Y 355.489,Z 217.283,A -85,B 0,C 180,E1 17353.957,E2 17353.957} C_VEL
LIN {X 0,Y 357.885,Z 219.505,A -85,B 0,C 180,E1 17353.674,E2 17353.674} C_VEL
LIN {X 0,Y 359.653,Z 219.219,A -85,B 0,C 180,E1 17353.549,E2 17353.549} C_VEL
LIN {X 0,Y 356.982,Z 302.492,A -85,B 0,C 180,E1 17351.58,E2 17351.58} C_VEL
LIN {X 0,Y 356.236,Z 319.264,A -85,B 0,C 180,E1 17350.875,E2 17350.875} C_VEL
LIN {X 0,Y 355.175,Z 334.75,A -85,B 0,C 180,E1 17349.912,E2 17349.912} C_VEL
LIN {X 0,Y 353.92,Z 349.081,A -85,B 0,C 180,E1 17348.722,E2 17348.722} C_VEL
LIN {X 0,Y 352.456,Z 363.041,A -85,B 0,C 180,E1 17347.217,E2 17347.217} C_VEL
LIN {X 0,Y 351.008,Z 375.508,A -85,B 0,C 180,E1 17345.496,E2 17345.496} C_VEL
LIN {X 0,Y 349.694,Z 386,A -85,B 0,C 180,E1 17343.692,E2 17343.692} C_VEL
LIN {X 0,Y 348.416,Z 395.801,A -85,B 0,C 180,E1 17341.55,E2 17341.55} C_VEL
LIN {X 0,Y 347.425,Z 403.615,A -85,B 0,C 180,E1 17339.373,E2 17339.373} C_VEL
LIN {X 0,Y 346.647,Z 410.07,A -85,B 0,C 180,E1 17336.965,E2 17336.965} C_VEL
LIN {X 0,Y 346.161,Z 414.744,A -85,B 0,C 180,E1 17334.508,E2 17334.508} C_VEL
LIN {X 0,Y 345.92,Z 417.827,A -85,B 0,C 180,E1 17331.789,E2 17331.789} C_VEL
LIN {X 0,Y 345.957,Z 418.862,A -85,B 0,C 180,E1 17329.218,E2 17329.218} C_VEL
LIN {X 0,Y 346.271,Z 418.111,A -85,B 0,C 180,E1 17326.588,E2 17326.588} C_VEL
LIN {X 0,Y 346.838,Z 415.637,A -85,B 0,C 180,E1 17324.125,E2 17324.125} C_VEL
LIN {X 0,Y 347.787,Z 411.115,A -85,B 0,C 180,E1 17321.513,E2 17321.513} C_VEL
LIN {X 0,Y 349.051,Z 404.789,A -85,B 0,C 180,E1 17319.065,E2 17319.065} C_VEL
LIN {X 0,Y 350.599,Z 396.896,A -85,B 0,C 180,E1 17316.791,E2 17316.791} C_VEL
LIN {X 0,Y 352.484,Z 386.723,A -85,B 0,C 180,E1 17314.564,E2 17314.564} C_VEL
LIN {X 0,Y 354.288,Z 376.161,A -85,B 0,C 180,E1 17312.753,E2 17312.753} C_VEL
LIN {X 0,Y 356.299,Z 363.193,A -85,B 0,C 180,E1 17310.994,E2 17310.994} C_VEL
LIN {X 0,Y 358.166,Z 349.073,A -85,B 0,C 180,E1 17309.511,E2 17309.511} C_VEL
LIN {X 0,Y 359.691,Z 335.233,A -85,B 0,C 180,E1 17308.382,E2 17308.382} C_VEL
LIN {X 0,Y 361.022,Z 319.145,A -85,B 0,C 180,E1 17307.416,E2 17307.416} C_VEL
LIN {X 0,Y 361.9,Z 303.223,A -85,B 0,C 180,E1 17306.766,E2 17306.766} C_VEL
LIN {X 0,Y 366.033,Z 209.965,A -85,B 0,C 180,E1 17304.371,E2 17304.371} C_VEL
LIN {X 0,Y 361.04,Z 180.696,A -85,B 0,C 180,E1 17302.931,E2 17302.931} C_VEL
LIN {X 0,Y 359.415,Z 171.875,A -85,B 0,C 180,E1 17302.404,E2 17302.404} C_VEL
LIN {X 0,Y 363.733,Z 145.504,A -85,B 0,C 180,E1 17297.932,E2 17297.932} C_VEL
LIN {X 0,Y 365.298,Z 136.487,A -85,B 0,C 180,E1 17296.375,E2 17296.375} C_VEL
LIN {X 0,Y 362.267,Z 123.558,A -85,B 0,C 180,E1 17293.243,E2 17293.243} C_VEL
LIN {X 0,Y 358.887,Z 112.012,A -85,B 0,C 180,E1 17290.109,E2 17290.109} C_VEL
LIN {X 0,Y 355.251,Z 101.27,A -85,B 0,C 180,E1 17286.789,E2 17286.789} C_VEL
LIN {X 0,Y 351.325,Z 91.106,A -85,B 0,C 180,E1 17283.1,E2 17283.1} C_VEL
LIN {X 0,Y 349.002,Z 86.193,A -85,B 0,C 180,E1 17280.969,E2 17280.969} C_VEL
LIN {X 0,Y 347.318,Z 82.377,A -85,B 0,C 180,E1 17279.176,E2 17279.176} C_VEL
LIN {X 0,Y 345.896,Z 78.792,A -85,B 0,C 180,E1 17277.184,E2 17277.184} C_VEL
LIN {X 0,Y 345.891,Z 78.714,A -85,B 0,C 180,E1 17273.027,E2 17273.027} C_VEL
LIN {X 0,Y 345.903,Z 78.712,A -85,B 0,C 180,E1 17268.833,E2 17268.833} C_VEL
LIN {X 0,Y 345.915,Z 78.709,A -85,B 0,C 180,E1 17264.578,E2 17264.578} C_VEL
LIN {X 0,Y 345.898,Z 78.711,A -85,B 0,C 180,E1 17260.409,E2 17260.409} C_VEL
LIN {X 0,Y 345.885,Z 78.715,A -85,B 0,C 180,E1 17256.309,E2 17256.309} C_VEL
LIN {X 0,Y 345.871,Z 78.716,A -85,B 0,C 180,E1 17252.075,E2 17252.075} C_VEL
LIN {X 0,Y 345.868,Z 78.714,A -85,B 0,C 180,E1 17247.865,E2 17247.865} C_VEL
LIN {X 0,Y 345.937,Z 79.026,A -85,B 0,C 180,E1 17246.777,E2 17246.777} C_VEL
LIN {X 0,Y 347.45,Z 82.541,A -85,B 0,C 180,E1 17245.064,E2 17245.064} C_VEL
LIN {X 0,Y 348.419,Z 84.5,A -85,B 0,C 180,E1 17244.168,E2 17244.168} C_VEL
LIN {X 0,Y 350.514,Z 88.8,A -85,B 0,C 180,E1 17242.379,E2 17242.379} C_VEL
LIN {X 0,Y 352.744,Z 93.728,A -85,B 0,C 180,E1 17240.585,E2 17240.585} C_VEL
LIN {X 0,Y 355.813,Z 100.376,A -85,B 0,C 180,E1 17238.373,E2 17238.373} C_VEL
LIN {X 0,Y 360.387,Z 111.759,A -85,B 0,C 180,E1 17235.195,E2 17235.195} C_VEL
LIN {X 0,Y 364.984,Z 124.553,A -85,B 0,C 180,E1 17232.158,E2 17232.158} C_VEL
LIN {X 0,Y 369.428,Z 139.116,A -85,B 0,C 180,E1 17229.206,E2 17229.206} C_VEL
LIN {X 0,Y 365.11,Z 162.988,A -85,B 0,C 180,E1 17226.292,E2 17226.292} C_VEL
LIN {X 0,Y 367.923,Z 189.672,A -85,B 0,C 180,E1 17225.317,E2 17225.317} C_VEL
LIN {X 0,Y 363.205,Z 351.05,A -85,B 0,C 180,E1 17222.054,E2 17222.054} C_VEL
LIN {X 0,Y 361.849,Z 369.396,A -85,B 0,C 180,E1 17221.42,E2 17221.42} C_VEL
LIN {X 0,Y 360.008,Z 386.628,A -85,B 0,C 180,E1 17220.548,E2 17220.548} C_VEL
LIN {X 0,Y 357.771,Z 403.801,A -85,B 0,C 180,E1 17219.372,E2 17219.372} C_VEL
LIN {X 0,Y 355.39,Z 419.953,A -85,B 0,C 180,E1 17217.944,E2 17217.944} C_VEL
LIN {X 0,Y 352.932,Z 435.426,A -85,B 0,C 180,E1 17216.229,E2 17216.229} C_VEL
LIN {X 0,Y 350.56,Z 449.904,A -85,B 0,C 180,E1 17214.251,E2 17214.251} C_VEL
LIN {X 0,Y 348.47,Z 463.038,A -85,B 0,C 180,E1 17212.063,E2 17212.063} C_VEL
LIN {X 0,Y 346.686,Z 475.415,A -85,B 0,C 180,E1 17209.546,E2 17209.546} C_VEL
LIN {X 0,Y 345.397,Z 486.321,A -85,B 0,C 180,E1 17206.828,E2 17206.828} C_VEL
LIN {X 0,Y 344.692,Z 495.675,A -85,B 0,C 180,E1 17203.932,E2 17203.932} C_VEL
LIN {X 0,Y 344.505,Z 503.04,A -85,B 0,C 180,E1 17201.044,E2 17201.044} C_VEL
LIN {X 0,Y 344.726,Z 508.591,A -85,B 0,C 180,E1 17198.172,E2 17198.172} C_VEL
LIN {X 0,Y 345.124,Z 512.433,A -85,B 0,C 180,E1 17195.321,E2 17195.321} C_VEL
LIN {X 0,Y 345.483,Z 514.632,A -85,B 0,C 180,E1 17192.489,E2 17192.489} C_VEL
LIN {X 0,Y 345.62,Z 515.212,A -85,B 0,C 180,E1 17189.836,E2 17189.836} C_VEL
LIN {X 0,Y 345.464,Z 514.34,A -85,B 0,C 180,E1 17187.181,E2 17187.181} C_VEL
LIN {X 0,Y 345.127,Z 512.004,A -85,B 0,C 180,E1 17184.515,E2 17184.515} C_VEL
LIN {X 0,Y 344.751,Z 507.844,A -85,B 0,C 180,E1 17181.663,E2 17181.663} C_VEL
LIN {X 0,Y 344.559,Z 501.813,A -85,B 0,C 180,E1 17178.761,E2 17178.761} C_VEL
LIN {X 0,Y 344.759,Z 493.992,A -85,B 0,C 180,E1 17175.902,E2 17175.902} C_VEL
LIN {X 0,Y 345.413,Z 484.573,A -85,B 0,C 180,E1 17173.176,E2 17173.176} C_VEL
LIN {X 0,Y 346.548,Z 473.7,A -85,B 0,C 180,E1 17170.624,E2 17170.624} C_VEL
LIN {X 0,Y 348.096,Z 461.375,A -85,B 0,C 180,E1 17168.253,E2 17168.253} C_VEL
LIN {X 0,Y 350.001,Z 447.526,A -85,B 0,C 180,E1 17166.07,E2 17166.07} C_VEL
LIN {X 0,Y 352.034,Z 433.021,A -85,B 0,C 180,E1 17164.204,E2 17164.204} C_VEL
LIN {X 0,Y 354.11,Z 417.628,A -85,B 0,C 180,E1 17162.599,E2 17162.599} C_VEL
LIN {X 0,Y 356.162,Z 400.985,A -85,B 0,C 180,E1 17161.222,E2 17161.222} C_VEL
LIN {X 0,Y 358.055,Z 383.186,A -85,B 0,C 180,E1 17160.104,E2 17160.104} C_VEL
LIN {X 0,Y 359.555,Z 365.298,A -85,B 0,C 180,E1 17159.296,E2 17159.296} C_VEL
LIN {X 0,Y 360.491,Z 346.43,A -85,B 0,C 180,E1 17158.744,E2 17158.744} C_VEL
LIN {X 0,Y 364.502,Z 176.147,A -85,B 0,C 180,E1 17155.406,E2 17155.406} C_VEL
LIN {X 0,Y 363.864,Z 157.164,A -85,B 0,C 180,E1 17154.883,E2 17154.883} C_VEL
LIN {X 0,Y 366.635,Z 128.866,A -85,B 0,C 180,E1 17152.939,E2 17152.939} C_VEL
LIN {X 0,Y 357.155,Z 104.791,A -85,B 0,C 180,E1 17150.091,E2 17150.091} C_VEL
LIN {X 0,Y 348.603,Z 85.323,A -85,B 0,C 180,E1 17147.487,E2 17147.487} C_VEL
LIN {X 0,Y 346.021,Z 79.273,A -85,B 0,C 180,E1 17146.601,E2 17146.601} C_VEL
LIN {X 0,Y 345.931,Z 78.713,A -85,B 0,C 180,E1 17146.268,E2 17146.268} C_VEL
LIN {X 0,Y 345.932,Z 78.705,A -85,B 0,C 180,E1 17142.031,E2 17142.031} C_VEL
LIN {X 0,Y 345.923,Z 78.704,A -85,B 0,C 180,E1 17137.789,E2 17137.789} C_VEL
LIN {X 0,Y 345.919,Z 78.709,A -85,B 0,C 180,E1 17133.509,E2 17133.509} C_VEL
LIN {X 0,Y 345.927,Z 78.706,A -85,B 0,C 180,E1 17129.208,E2 17129.208} C_VEL
LIN {X 0,Y 345.93,Z 78.707,A -85,B 0,C 180,E1 17124.96,E2 17124.96} C_VEL
LIN {X 0,Y 345.935,Z 78.708,A -85,B 0,C 180,E1 17120.824,E2 17120.824} C_VEL
LIN {X 0,Y 345.93,Z 78.709,A -85,B 0,C 180,E1 17116.627,E2 17116.627} C_VEL
LIN {X 0,Y 345.921,Z 78.707,A -85,B 0,C 180,E1 17112.52,E2 17112.52} C_VEL
LIN {X 0,Y 345.912,Z 78.702,A -85,B 0,C 180,E1 17108.309,E2 17108.309} C_VEL
LIN {X 0,Y 345.906,Z 78.698,A -85,B 0,C 180,E1 17103.978,E2 17103.978} C_VEL
LIN {X 0,Y 345.909,Z 78.693,A -85,B 0,C 180,E1 17099.834,E2 17099.834} C_VEL
LIN {X 0,Y 345.922,Z 78.697,A -85,B 0,C 180,E1 17095.524,E2 17095.524} C_VEL
LIN {X 0,Y 345.929,Z 78.699,A -85,B 0,C 180,E1 17091.289,E2 17091.289} C_VEL
LIN {X 0,Y 345.91,Z 78.701,A -85,B 0,C 180,E1 17086.97,E2 17086.97} C_VEL
LIN {X 0,Y 345.902,Z 78.703,A -85,B 0,C 180,E1 17082.852,E2 17082.852} C_VEL
LIN {X 0,Y 345.895,Z 78.7,A -85,B 0,C 180,E1 17078.552,E2 17078.552} C_VEL
LIN {X 0,Y 345.902,Z 78.695,A -85,B 0,C 180,E1 17074.304,E2 17074.304} C_VEL
LIN {X 0,Y 345.912,Z 78.679,A -85,B 0,C 180,E1 17070.125,E2 17070.125} C_VEL
LIN {X 0,Y 345.924,Z 78.699,A -85,B 0,C 180,E1 17065.893,E2 17065.893} C_VEL
LIN {X 0,Y 345.906,Z 78.713,A -85,B 0,C 180,E1 17061.564,E2 17061.564} C_VEL
LIN {X 0,Y 345.894,Z 78.709,A -85,B 0,C 180,E1 17057.435,E2 17057.435} C_VEL
LIN {X 0,Y 345.928,Z 78.782,A -85,B 0,C 180,E1 17056.203,E2 17056.203} C_VEL
LIN {X 0,Y 346.192,Z 80.024,A -85,B 0,C 180,E1 17055.889,E2 17055.889} C_VEL
LIN {X 0,Y 352.166,Z 94.877,A -85,B 0,C 180,E1 17053.26,E2 17053.26} C_VEL
LIN {X 0,Y 357.543,Z 111.13,A -85,B 0,C 180,E1 17050.614,E2 17050.614} C_VEL
LIN {X 0,Y 360.252,Z 121.708,A -85,B 0,C 180,E1 17049.001,E2 17049.001} C_VEL
LIN {X 0,Y 359,Z 157.316,A -85,B 0,C 180,E1 17044.753,E2 17044.753} C_VEL
LIN {X 0,Y 357.848,Z 194.033,A -85,B 0,C 180,E1 17040.471,E2 17040.471} C_VEL
LIN {X 0,Y 357.701,Z 204.18,A -85,B 0,C 180,E1 17039.384,E2 17039.384} C_VEL
LIN {X 0,Y 358.329,Z 209.508,A -85,B 0,C 180,E1 17039.216,E2 17039.216} C_VEL
LIN {X 0,Y 356.323,Z 309.042,A -85,B 0,C 180,E1 17037.192,E2 17037.192} C_VEL
LIN {X 0,Y 356.255,Z 324.821,A -85,B 0,C 180,E1 17036.704,E2 17036.704} C_VEL
LIN {X 0,Y 355.721,Z 339.889,A -85,B 0,C 180,E1 17035.913,E2 17035.913} C_VEL
LIN {X 0,Y 354.777,Z 354.106,A -85,B 0,C 180,E1 17034.828,E2 17034.828} C_VEL
LIN {X 0,Y 353.643,Z 366.306,A -85,B 0,C 180,E1 17033.58,E2 17033.58} C_VEL
LIN {X 0,Y 352.376,Z 377.706,A -85,B 0,C 180,E1 17032.082,E2 17032.082} C_VEL
LIN {X 0,Y 350.862,Z 388.949,A -85,B 0,C 180,E1 17030.169,E2 17030.169} C_VEL
LIN {X 0,Y 349.387,Z 398.629,A -85,B 0,C 180,E1 17028.001,E2 17028.001} C_VEL
LIN {X 0,Y 348.111,Z 406.411,A -85,B 0,C 180,E1 17025.662,E2 17025.662} C_VEL
LIN {X 0,Y 347.148,Z 411.982,A -85,B 0,C 180,E1 17023.32,E2 17023.32} C_VEL
LIN {X 0,Y 346.478,Z 415.706,A -85,B 0,C 180,E1 17020.978,E2 17020.978} C_VEL
LIN {X 0,Y 346.04,Z 417.863,A -85,B 0,C 180,E1 17018.473,E2 17018.473} C_VEL
LIN {X 0,Y 345.837,Z 418.156,A -85,B 0,C 180,E1 17015.806,E2 17015.806} C_VEL
LIN {X 0,Y 345.894,Z 416.42,A -85,B 0,C 180,E1 17013.147,E2 17013.147} C_VEL
LIN {X 0,Y 346.188,Z 412.896,A -85,B 0,C 180,E1 17010.661,E2 17010.661} C_VEL
LIN {X 0,Y 346.691,Z 407.811,A -85,B 0,C 180,E1 17008.346,E2 17008.346} C_VEL
LIN {X 0,Y 347.384,Z 401.317,A -85,B 0,C 180,E1 17006.203,E2 17006.203} C_VEL
LIN {X 0,Y 348.304,Z 392.708,A -85,B 0,C 180,E1 17004.067,E2 17004.067} C_VEL
LIN {X 0,Y 349.263,Z 383.354,A -85,B 0,C 180,E1 17002.266,E2 17002.266} C_VEL
LIN {X 0,Y 350.315,Z 372.019,A -85,B 0,C 180,E1 17000.553,E2 17000.553} C_VEL
LIN {X 0,Y 351.265,Z 359.47,A -85,B 0,C 180,E1 16999.088,E2 16999.088} C_VEL
LIN {X 0,Y 352.108,Z 345.503,A -85,B 0,C 180,E1 16997.869,E2 16997.869} C_VEL
LIN {X 0,Y 352.63,Z 331.354,A -85,B 0,C 180,E1 16996.982,E2 16996.982} C_VEL
LIN {X 0,Y 352.806,Z 316.772,A -85,B 0,C 180,E1 16996.379,E2 16996.379} C_VEL
LIN {X 0,Y 352.754,Z 298.07,A -85,B 0,C 180,E1 16995.943,E2 16995.943} C_VEL
LIN {X 0,Y 351.845,Z 290.459,A -85,B 0,C 180,E1 16995.733,E2 16995.733} C_VEL
LIN {X 0,Y 346.297,Z 270.468,A -85,B 0,C 180,E1 16994.989,E2 16994.989} C_VEL
LIN {X 0,Y 345.749,Z 263.925,A -85,B 0,C 180,E1 16994.815,E2 16994.815} C_VEL
LIN {X 0,Y 346.259,Z 244.39,A -85,B 0,C 180,E1 16994.367,E2 16994.367} C_VEL
LIN {X 0,Y 346.928,Z 241.315,A -85,B 0,C 180,E1 16994.109,E2 16994.109} C_VEL
LIN {X 0,Y 347.79,Z 240.875,A -85,B 0,C 180,E1 16993.914,E2 16993.914} C_VEL
LIN {X 0,Y 349.479,Z 242.827,A -85,B 0,C 180,E1 16993.716,E2 16993.716} C_VEL
LIN {X 0,Y 351.282,Z 242.724,A -85,B 0,C 180,E1 16993.58,E2 16993.58} C_VEL
LIN {X 0,Y 351.597,Z 242.731,A -85,B 0,C 180,E1 16993.556,E2 16993.556} C_VEL
LIN {X 0,Y 349.586,Z 303.604,A -85,B 0,C 180,E1 16992.056,E2 16992.056} C_VEL
LIN {X 0,Y 348.805,Z 320.19,A -85,B 0,C 180,E1 16991.338,E2 16991.338} C_VEL
LIN {X 0,Y 347.678,Z 335.865,A -85,B 0,C 180,E1 16990.337,E2 16990.337} C_VEL
LIN {X 0,Y 346.356,Z 350.201,A -85,B 0,C 180,E1 16989.112,E2 16989.112} C_VEL
LIN {X 0,Y 344.85,Z 363.965,A -85,B 0,C 180,E1 16987.596,E2 16987.596} C_VEL
LIN {X 0,Y 343.372,Z 376.154,A -85,B 0,C 180,E1 16985.881,E2 16985.881} C_VEL
LIN {X 0,Y 341.881,Z 387.518,A -85,B 0,C 180,E1 16983.878,E2 16983.878} C_VEL
LIN {X 0,Y 340.511,Z 397.6,A -85,B 0,C 180,E1 16981.595,E2 16981.595} C_VEL
LIN {X 0,Y 339.475,Z 405.348,A -85,B 0,C 180,E1 16979.321,E2 16979.321} C_VEL
LIN {X 0,Y 338.706,Z 411.577,A -85,B 0,C 180,E1 16976.898,E2 16976.898} C_VEL
LIN {X 0,Y 338.214,Z 416.099,A -85,B 0,C 180,E1 16974.38,E2 16974.38} C_VEL
LIN {X 0,Y 337.995,Z 418.916,A -85,B 0,C 180,E1 16971.81,E2 16971.81} C_VEL
LIN {X 0,Y 338.039,Z 419.993,A -85,B 0,C 180,E1 16969.18,E2 16969.18} C_VEL
LIN {X 0,Y 338.376,Z 419.28,A -85,B 0,C 180,E1 16966.489,E2 16966.489} C_VEL
LIN {X 0,Y 339.012,Z 416.745,A -85,B 0,C 180,E1 16963.876,E2 16963.876} C_VEL
LIN {X 0,Y 340.041,Z 412.203,A -85,B 0,C 180,E1 16961.198,E2 16961.198} C_VEL
LIN {X 0,Y 341.411,Z 405.803,A -85,B 0,C 180,E1 16958.674,E2 16958.674} C_VEL
LIN {X 0,Y 343.005,Z 398.206,A -85,B 0,C 180,E1 16956.433,E2 16956.433} C_VEL
LIN {X 0,Y 344.939,Z 388.389,A -85,B 0,C 180,E1 16954.218,E2 16954.218} C_VEL
LIN {X 0,Y 346.85,Z 378.035,A -85,B 0,C 180,E1 16952.367,E2 16952.367} C_VEL
LIN {X 0,Y 348.962,Z 365.256,A -85,B 0,C 180,E1 16950.57,E2 16950.57} C_VEL
LIN {X 0,Y 350.777,Z 352.684,A -85,B 0,C 180,E1 16949.172,E2 16949.172} C_VEL
LIN {X 0,Y 352.61,Z 337.25,A -85,B 0,C 180,E1 16947.847,E2 16947.847} C_VEL
LIN {X 0,Y 354.011,Z 321.703,A -85,B 0,C 180,E1 16946.866,E2 16946.866} C_VEL
LIN {X 0,Y 355.021,Z 305.374,A -85,B 0,C 180,E1 16946.153,E2 16946.153} C_VEL
LIN {X 0,Y 359.424,Z 211.269,A -85,B 0,C 180,E1 16943.675,E2 16943.675} C_VEL
LIN {X 0,Y 354.587,Z 182.423,A -85,B 0,C 180,E1 16942.201,E2 16942.201} C_VEL
LIN {X 0,Y 352.634,Z 171.796,A -85,B 0,C 180,E1 16941.563,E2 16941.563} C_VEL
LIN {X 0,Y 357.229,Z 145.468,A -85,B 0,C 180,E1 16937.007,E2 16937.007} C_VEL
LIN {X 0,Y 358.268,Z 139.535,A -85,B 0,C 180,E1 16935.956,E2 16935.956} C_VEL
LIN {X 0,Y 355.379,Z 127.031,A -85,B 0,C 180,E1 16932.843,E2 16932.843} C_VEL
LIN {X 0,Y 352.128,Z 115.661,A -85,B 0,C 180,E1 16929.645,E2 16929.645} C_VEL
LIN {X 0,Y 348.754,Z 105.623,A -85,B 0,C 180,E1 16926.42,E2 16926.42} C_VEL
LIN {X 0,Y 345.332,Z 96.418,A -85,B 0,C 180,E1 16922.988,E2 16922.988} C_VEL
LIN {X 0,Y 342.95,Z 91.227,A -85,B 0,C 180,E1 16920.669,E2 16920.669} C_VEL
LIN {X 0,Y 341.645,Z 88.029,A -85,B 0,C 180,E1 16919.162,E2 16919.162} C_VEL
LIN {X 0,Y 339.529,Z 83.542,A -85,B 0,C 180,E1 16916.663,E2 16916.663} C_VEL
LIN {X 0,Y 337.977,Z 79.808,A -85,B 0,C 180,E1 16914.142,E2 16914.142} C_VEL
LIN {X 0,Y 337.948,Z 79.697,A -85,B 0,C 180,E1 16909.947,E2 16909.947} C_VEL
LIN {X 0,Y 337.937,Z 79.698,A -85,B 0,C 180,E1 16905.61,E2 16905.61} C_VEL
LIN {X 0,Y 337.942,Z 79.696,A -85,B 0,C 180,E1 16901.365,E2 16901.365} C_VEL
LIN {X 0,Y 337.952,Z 79.696,A -85,B 0,C 180,E1 16897.197,E2 16897.197} C_VEL
LIN {X 0,Y 337.969,Z 79.695,A -85,B 0,C 180,E1 16892.897,E2 16892.897} C_VEL
LIN {X 0,Y 337.978,Z 80.019,A -85,B 0,C 180,E1 16889.849,E2 16889.849} C_VEL
LIN {X 0,Y 339.841,Z 83.958,A -85,B 0,C 180,E1 16887.425,E2 16887.425} C_VEL
LIN {X 0,Y 340.754,Z 86.104,A -85,B 0,C 180,E1 16886.319,E2 16886.319} C_VEL
LIN {X 0,Y 342.713,Z 89.775,A -85,B 0,C 180,E1 16884.487,E2 16884.487} C_VEL
LIN {X 0,Y 345.08,Z 95.021,A -85,B 0,C 180,E1 16882.312,E2 16882.312} C_VEL
LIN {X 0,Y 347.083,Z 99.426,A -85,B 0,C 180,E1 16880.672,E2 16880.672} C_VEL
LIN {X 0,Y 350.035,Z 106.064,A -85,B 0,C 180,E1 16878.452,E2 16878.452} C_VEL
LIN {X 0,Y 354.347,Z 116.927,A -85,B 0,C 180,E1 16875.364,E2 16875.364} C_VEL
LIN {X 0,Y 358.652,Z 129.274,A -85,B 0,C 180,E1 16872.373,E2 16872.373} C_VEL
LIN {X 0,Y 362.569,Z 142.511,A -85,B 0,C 180,E1 16869.626,E2 16869.626} C_VEL
LIN {X 0,Y 358.524,Z 163.318,A -85,B 0,C 180,E1 16867.058,E2 16867.058} C_VEL
LIN {X 0,Y 361.347,Z 190.51,A -85,B 0,C 180,E1 16866.025,E2 16866.025} C_VEL
LIN {X 0,Y 356.966,Z 333.643,A -85,B 0,C 180,E1 16863.104,E2 16863.104} C_VEL
LIN {X 0,Y 356.113,Z 354.812,A -85,B 0,C 180,E1 16862.598,E2 16862.598} C_VEL
LIN {X 0,Y 354.526,Z 373.128,A -85,B 0,C 180,E1 16861.888,E2 16861.888} C_VEL
LIN {X 0,Y 352.406,Z 390.682,A -85,B 0,C 180,E1 16860.901,E2 16860.901} C_VEL
LIN {X 0,Y 349.986,Z 407.633,A -85,B 0,C 180,E1 16859.62,E2 16859.62} C_VEL
LIN {X 0,Y 347.406,Z 423.704,A -85,B 0,C 180,E1 16858.072,E2 16858.072} C_VEL
LIN {X 0,Y 344.712,Z 439.498,A -85,B 0,C 180,E1 16856.161,E2 16856.161} C_VEL
LIN {X 0,Y 342.261,Z 453.627,A -85,B 0,C 180,E1 16854.05,E2 16854.05} C_VEL
LIN {X 0,Y 340.147,Z 466.314,A -85,B 0,C 180,E1 16851.74,E2 16851.74} C_VEL
LIN {X 0,Y 338.424,Z 478.038,A -85,B 0,C 180,E1 16849.145,E2 16849.145} C_VEL
LIN {X 0,Y 337.227,Z 488.266,A -85,B 0,C 180,E1 16846.361,E2 16846.361} C_VEL
LIN {X 0,Y 336.624,Z 496.977,A -85,B 0,C 180,E1 16843.397,E2 16843.397} C_VEL
LIN {X 0,Y 336.541,Z 503.769,A -85,B 0,C 180,E1 16840.443,E2 16840.443} C_VEL
LIN {X 0,Y 336.871,Z 509.039,A -85,B 0,C 180,E1 16837.334,E2 16837.334} C_VEL
LIN {X 0,Y 337.31,Z 512.297,A -85,B 0,C 180,E1 16834.421,E2 16834.421} C_VEL
LIN {X 0,Y 337.636,Z 513.914,A -85,B 0,C 180,E1 16831.528,E2 16831.528} C_VEL
LIN {X 0,Y 337.667,Z 513.944,A -85,B 0,C 180,E1 16828.814,E2 16828.814} C_VEL
LIN {X 0,Y 337.409,Z 512.492,A -85,B 0,C 180,E1 16826.093,E2 16826.093} C_VEL
LIN {X 0,Y 336.995,Z 509.292,A -85,B 0,C 180,E1 16823.186,E2 16823.186} C_VEL
LIN {X 0,Y 336.65,Z 504.354,A -85,B 0,C 180,E1 16820.255,E2 16820.255} C_VEL
LIN {X 0,Y 336.624,Z 497.568,A -85,B 0,C 180,E1 16817.304,E2 16817.304} C_VEL
LIN {X 0,Y 337.021,Z 489.318,A -85,B 0,C 180,E1 16814.515,E2 16814.515} C_VEL
LIN {X 0,Y 337.965,Z 479.06,A -85,B 0,C 180,E1 16811.744,E2 16811.744} C_VEL
LIN {X 0,Y 339.418,Z 467.055,A -85,B 0,C 180,E1 16809.12,E2 16809.12} C_VEL
LIN {X 0,Y 341.234,Z 454.01,A -85,B 0,C 180,E1 16806.792,E2 16806.792} C_VEL
LIN {X 0,Y 343.28,Z 439.995,A -85,B 0,C 180,E1 16804.743,E2 16804.743} C_VEL
LIN {X 0,Y 345.426,Z 425.136,A -85,B 0,C 180,E1 16802.973,E2 16802.973} C_VEL
LIN {X 0,Y 347.668,Z 408.641,A -85,B 0,C 180,E1 16801.397,E2 16801.397} C_VEL
LIN {X 0,Y 349.718,Z 391.428,A -85,B 0,C 180,E1 16800.126,E2 16800.126} C_VEL
LIN {X 0,Y 351.491,Z 373.695,A -85,B 0,C 180,E1 16799.155,E2 16799.155} C_VEL
LIN {X 0,Y 352.796,Z 355.332,A -85,B 0,C 180,E1 16798.464,E2 16798.464} C_VEL
LIN {X 0,Y 353.553,Z 329.379,A -85,B 0,C 180,E1 16797.887,E2 16797.887} C_VEL
LIN {X 0,Y 357.336,Z 176.097,A -85,B 0,C 180,E1 16794.822,E2 16794.822} C_VEL
LIN {X 0,Y 356.741,Z 157.279,A -85,B 0,C 180,E1 16794.293,E2 16794.293} C_VEL
LIN {X 0,Y 359.335,Z 131.172,A -85,B 0,C 180,E1 16792.458,E2 16792.458} C_VEL
LIN {X 0,Y 350.111,Z 107.668,A -85,B 0,C 180,E1 16789.591,E2 16789.591} C_VEL
LIN {X 0,Y 341.093,Z 87.044,A -85,B 0,C 180,E1 16786.755,E2 16786.755} C_VEL
LIN {X 0,Y 338.065,Z 80.194,A -85,B 0,C 180,E1 16785.703,E2 16785.703} C_VEL
LIN {X 0,Y 337.985,Z 79.695,A -85,B 0,C 180,E1 16785.234,E2 16785.234} C_VEL
LIN {X 0,Y 338.002,Z 79.689,A -85,B 0,C 180,E1 16780.778,E2 16780.778} C_VEL
LIN {X 0,Y 337.991,Z 79.697,A -85,B 0,C 180,E1 16776.428,E2 16776.428} C_VEL
LIN {X 0,Y 337.988,Z 79.688,A -85,B 0,C 180,E1 16772.173,E2 16772.173} C_VEL
LIN {X 0,Y 337.979,Z 79.686,A -85,B 0,C 180,E1 16767.867,E2 16767.867} C_VEL
LIN {X 0,Y 337.978,Z 79.683,A -85,B 0,C 180,E1 16763.501,E2 16763.501} C_VEL
LIN {X 0,Y 337.989,Z 79.683,A -85,B 0,C 180,E1 16759.169,E2 16759.169} C_VEL
LIN {X 0,Y 337.997,Z 79.684,A -85,B 0,C 180,E1 16754.913,E2 16754.913} C_VEL
LIN {X 0,Y 337.98,Z 79.688,A -85,B 0,C 180,E1 16750.569,E2 16750.569} C_VEL
LIN {X 0,Y 337.97,Z 79.694,A -85,B 0,C 180,E1 16746.284,E2 16746.284} C_VEL
LIN {X 0,Y 337.971,Z 79.696,A -85,B 0,C 180,E1 16741.865,E2 16741.865} C_VEL
LIN {X 0,Y 337.979,Z 79.696,A -85,B 0,C 180,E1 16737.626,E2 16737.626} C_VEL
LIN {X 0,Y 337.997,Z 79.694,A -85,B 0,C 180,E1 16733.204,E2 16733.204} C_VEL
LIN {X 0,Y 337.971,Z 79.696,A -85,B 0,C 180,E1 16728.913,E2 16728.913} C_VEL
LIN {X 0,Y 337.959,Z 79.699,A -85,B 0,C 180,E1 16724.557,E2 16724.557} C_VEL
LIN {X 0,Y 337.968,Z 79.698,A -85,B 0,C 180,E1 16720.177,E2 16720.177} C_VEL
LIN {X 0,Y 337.978,Z 79.655,A -85,B 0,C 180,E1 16715.904,E2 16715.904} C_VEL
LIN {X 0,Y 337.991,Z 79.685,A -85,B 0,C 180,E1 16711.75,E2 16711.75} C_VEL
LIN {X 0,Y 337.97,Z 79.696,A -85,B 0,C 180,E1 16707.47,E2 16707.47} C_VEL
LIN {X 0,Y 337.955,Z 79.683,A -85,B 0,C 180,E1 16703.296,E2 16703.296} C_VEL
LIN {X 0,Y 337.947,Z 79.686,A -85,B 0,C 180,E1 16698.974,E2 16698.974} C_VEL
LIN {X 0,Y 337.986,Z 79.971,A -85,B 0,C 180,E1 16697.066,E2 16697.066} C_VEL
LIN {X 0,Y 343.487,Z 93.611,A -85,B 0,C 180,E1 16694.506,E2 16694.506} C_VEL
LIN {X 0,Y 348.987,Z 109.196,A -85,B 0,C 180,E1 16691.848,E2 16691.848} C_VEL
LIN {X 0,Y 353.209,Z 124.426,A -85,B 0,C 180,E1 16689.445,E2 16689.445} C_VEL
LIN {X 0,Y 351.87,Z 159.46,A -85,B 0,C 180,E1 16685.226,E2 16685.226} C_VEL
LIN {X 0,Y 350.674,Z 195.757,A -85,B 0,C 180,E1 16680.972,E2 16680.972} C_VEL
LIN {X 0,Y 350.514,Z 205.243,A -85,B 0,C 180,E1 16679.949,E2 16679.949} C_VEL
LIN {X 0,Y 351.151,Z 210.524,A -85,B 0,C 180,E1 16679.776,E2 16679.776} C_VEL
LIN {X 0,Y 349.039,Z 309.493,A -85,B 0,C 180,E1 16677.724,E2 16677.724} C_VEL
LIN {X 0,Y 348.968,Z 325.571,A -85,B 0,C 180,E1 16677.226,E2 16677.226} C_VEL
LIN {X 0,Y 348.396,Z 340.881,A -85,B 0,C 180,E1 16676.411,E2 16676.411} C_VEL
LIN {X 0,Y 347.404,Z 355.07,A -85,B 0,C 180,E1 16675.31,E2 16675.31} C_VEL
LIN {X 0,Y 346.202,Z 367.378,A -85,B 0,C 180,E1 16674.028,E2 16674.028} C_VEL
LIN {X 0,Y 344.864,Z 378.785,A -85,B 0,C 180,E1 16672.5,E2 16672.5} C_VEL
LIN {X 0,Y 343.33,Z 389.594,A -85,B 0,C 180,E1 16670.631,E2 16670.631} C_VEL
LIN {X 0,Y 341.866,Z 398.706,A -85,B 0,C 180,E1 16668.588,E2 16668.588} C_VEL
LIN {X 0,Y 340.655,Z 405.767,A -85,B 0,C 180,E1 16666.54,E2 16666.54} C_VEL
LIN {X 0,Y 339.554,Z 411.886,A -85,B 0,C 180,E1 16664.145,E2 16664.145} C_VEL
LIN {X 0,Y 338.719,Z 416.269,A -85,B 0,C 180,E1 16661.578,E2 16661.578} C_VEL
LIN {X 0,Y 338.189,Z 418.706,A -85,B 0,C 180,E1 16659.014,E2 16659.014} C_VEL
LIN {X 0,Y 337.934,Z 419.343,A -85,B 0,C 180,E1 16656.454,E2 16656.454} C_VEL
LIN {X 0,Y 337.925,Z 418.217,A -85,B 0,C 180,E1 16653.901,E2 16653.901} C_VEL
LIN {X 0,Y 338.182,Z 415.005,A -85,B 0,C 180,E1 16651.185,E2 16651.185} C_VEL
LIN {X 0,Y 338.689,Z 409.962,A -85,B 0,C 180,E1 16648.645,E2 16648.645} C_VEL
LIN {X 0,Y 339.366,Z 403.789,A -85,B 0,C 180,E1 16646.452,E2 16646.452} C_VEL
LIN {X 0,Y 340.287,Z 395.649,A -85,B 0,C 180,E1 16644.265,E2 16644.265} C_VEL
LIN {X 0,Y 341.352,Z 385.886,A -85,B 0,C 180,E1 16642.255,E2 16642.255} C_VEL
LIN {X 0,Y 342.489,Z 374.322,A -85,B 0,C 180,E1 16640.42,E2 16640.42} C_VEL
LIN {X 0,Y 343.474,Z 362.099,A -85,B 0,C 180,E1 16638.922,E2 16638.922} C_VEL
LIN {X 0,Y 344.299,Z 349.769,A -85,B 0,C 180,E1 16637.76,E2 16637.76} C_VEL
LIN {X 0,Y 344.952,Z 335.362,A -85,B 0,C 180,E1 16636.762,E2 16636.762} C_VEL
LIN {X 0,Y 345.213,Z 319.874,A -85,B 0,C 180,E1 16636.053,E2 16636.053} C_VEL
LIN {X 0,Y 345.226,Z 292.252,A -85,B 0,C 180,E1 16635.397,E2 16635.397} C_VEL
LIN {X 0,Y 345.749,Z 263.925,A -85,B 0,C 180,E1 16634.815,E2 16634.815} C_VEL
LIN {X 0,Y 345.522,Z 263.966,A -85,B 0,C 180,E1 16634.618,E2 16634.618} C_VEL
LIN {X 0,Y 345.048,Z 266.192,A -85,B 0,C 180,E1 16634.286,E2 16634.286} C_VEL
LIN {X 0,Y 344.317,Z 271.772,A -85,B 0,C 180,E1 16633.842,E2 16633.842} C_VEL
LIN {X 0,Y 342.748,Z 290.77,A -85,B 0,C 180,E1 16632.995,E2 16632.995} C_VEL
LIN {X 0,Y 342.459,Z 297.218,A -85,B 0,C 180,E1 16632.786,E2 16632.786} C_VEL
LIN {X 0,Y 341.765,Z 314.598,A -85,B 0,C 180,E1 16632.149,E2 16632.149} C_VEL
LIN {X 0,Y 340.68,Z 331.006,A -85,B 0,C 180,E1 16631.209,E2 16631.209} C_VEL
LIN {X 0,Y 339.362,Z 345.923,A -85,B 0,C 180,E1 16630.031,E2 16630.031} C_VEL
LIN {X 0,Y 337.804,Z 360.276,A -85,B 0,C 180,E1 16628.553,E2 16628.553} C_VEL
LIN {X 0,Y 336.176,Z 373.534,A -85,B 0,C 180,E1 16626.786,E2 16626.786} C_VEL
LIN {X 0,Y 334.634,Z 384.947,A -85,B 0,C 180,E1 16624.87,E2 16624.87} C_VEL
LIN {X 0,Y 333.17,Z 395.345,A -85,B 0,C 180,E1 16622.663,E2 16622.663} C_VEL
LIN {X 0,Y 331.994,Z 403.636,A -85,B 0,C 180,E1 16620.401,E2 16620.401} C_VEL
LIN {X 0,Y 331.054,Z 410.695,A -85,B 0,C 180,E1 16617.888,E2 16617.888} C_VEL
LIN {X 0,Y 330.436,Z 415.815,A -85,B 0,C 180,E1 16615.328,E2 16615.328} C_VEL
LIN {X 0,Y 330.118,Z 419.256,A -85,B 0,C 180,E1 16612.716,E2 16612.716} C_VEL
LIN {X 0,Y 330.072,Z 420.935,A -85,B 0,C 180,E1 16610.032,E2 16610.032} C_VEL
LIN {X 0,Y 330.325,Z 420.904,A -85,B 0,C 180,E1 16607.31,E2 16607.31} C_VEL
LIN {X 0,Y 330.857,Z 419.154,A -85,B 0,C 180,E1 16604.75,E2 16604.75} C_VEL
LIN {X 0,Y 331.801,Z 415.417,A -85,B 0,C 180,E1 16601.989,E2 16601.989} C_VEL
LIN {X 0,Y 333.028,Z 410.159,A -85,B 0,C 180,E1 16599.502,E2 16599.502} C_VEL
LIN {X 0,Y 334.628,Z 403.16,A -85,B 0,C 180,E1 16597.08,E2 16597.08} C_VEL
LIN {X 0,Y 336.538,Z 394.353,A -85,B 0,C 180,E1 16594.781,E2 16594.781} C_VEL
LIN {X 0,Y 338.701,Z 383.762,A -85,B 0,C 180,E1 16592.627,E2 16592.627} C_VEL
LIN {X 0,Y 340.946,Z 371.455,A -85,B 0,C 180,E1 16590.683,E2 16590.683} C_VEL
LIN {X 0,Y 342.957,Z 359.087,A -85,B 0,C 180,E1 16589.136,E2 16589.136} C_VEL
LIN {X 0,Y 344.927,Z 344.659,A -85,B 0,C 180,E1 16587.727,E2 16587.727} C_VEL
LIN {X 0,Y 346.521,Z 330.249,A -85,B 0,C 180,E1 16586.65,E2 16586.65} C_VEL
LIN {X 0,Y 347.877,Z 313.337,A -85,B 0,C 180,E1 16585.742,E2 16585.742} C_VEL
LIN {X 0,Y 348.797,Z 294.377,A -85,B 0,C 180,E1 16585.109,E2 16585.109} C_VEL
LIN {X 0,Y 352.897,Z 212.563,A -85,B 0,C 180,E1 16582.946,E2 16582.946} C_VEL
LIN {X 0,Y 348.075,Z 183.308,A -85,B 0,C 180,E1 16581.396,E2 16581.396} C_VEL
LIN {X 0,Y 345.948,Z 171.837,A -85,B 0,C 180,E1 16580.691,E2 16580.691} C_VEL
LIN {X 0,Y 350.747,Z 145.936,A -85,B 0,C 180,E1 16576.121,E2 16576.121} C_VEL
LIN {X 0,Y 351.295,Z 142.662,A -85,B 0,C 180,E1 16575.519,E2 16575.519} C_VEL
LIN {X 0,Y 348.438,Z 130.014,A -85,B 0,C 180,E1 16572.26,E2 16572.26} C_VEL
LIN {X 0,Y 345.301,Z 118.849,A -85,B 0,C 180,E1 16568.996,E2 16568.996} C_VEL
LIN {X 0,Y 342.15,Z 109.543,A -85,B 0,C 180,E1 16565.871,E2 16565.871} C_VEL
LIN {X 0,Y 339.174,Z 101.33,A -85,B 0,C 180,E1 16562.704,E2 16562.704} C_VEL
LIN {X 0,Y 336.907,Z 96.217,A -85,B 0,C 180,E1 16560.34,E2 16560.34} C_VEL
LIN {X 0,Y 335.64,Z 93.153,A -85,B 0,C 180,E1 16558.805,E2 16558.805} C_VEL
LIN {X 0,Y 333.896,Z 89.196,A -85,B 0,C 180,E1 16556.567,E2 16556.567} C_VEL
LIN {X 0,Y 331.952,Z 85.022,A -85,B 0,C 180,E1 16553.711,E2 16553.711} C_VEL
LIN {X 0,Y 330.022,Z 80.827,A -85,B 0,C 180,E1 16549.703,E2 16549.703} C_VEL
LIN {X 0,Y 330.007,Z 80.688,A -85,B 0,C 180,E1 16545.256,E2 16545.256} C_VEL
LIN {X 0,Y 330.026,Z 80.685,A -85,B 0,C 180,E1 16540.901,E2 16540.901} C_VEL
LIN {X 0,Y 330.026,Z 80.687,A -85,B 0,C 180,E1 16536.617,E2 16536.617} C_VEL
LIN {X 0,Y 330.053,Z 81.039,A -85,B 0,C 180,E1 16534.233,E2 16534.233} C_VEL
LIN {X 0,Y 332.616,Z 86.085,A -85,B 0,C 180,E1 16529.867,E2 16529.867} C_VEL
LIN {X 0,Y 335.013,Z 90.979,A -85,B 0,C 180,E1 16526.896,E2 16526.896} C_VEL
LIN {X 0,Y 337.147,Z 95.492,A -85,B 0,C 180,E1 16524.643,E2 16524.643} C_VEL
LIN {X 0,Y 339.278,Z 100.229,A -85,B 0,C 180,E1 16522.621,E2 16522.621} C_VEL
LIN {X 0,Y 342.21,Z 106.579,A -85,B 0,C 180,E1 16520.213,E2 16520.213} C_VEL
LIN {X 0,Y 346.437,Z 117.102,A -85,B 0,C 180,E1 16516.903,E2 16516.903} C_VEL
LIN {X 0,Y 350.72,Z 129.182,A -85,B 0,C 180,E1 16513.723,E2 16513.723} C_VEL
LIN {X 0,Y 354.68,Z 141.999,A -85,B 0,C 180,E1 16510.846,E2 16510.846} C_VEL
LIN {X 0,Y 355.599,Z 145.851,A -85,B 0,C 180,E1 16510.084,E2 16510.084} C_VEL
LIN {X 0,Y 352.001,Z 163.514,A -85,B 0,C 180,E1 16507.863,E2 16507.863} C_VEL
LIN {X 0,Y 354.865,Z 191.234,A -85,B 0,C 180,E1 16506.768,E2 16506.768} C_VEL
LIN {X 0,Y 350.113,Z 336.793,A -85,B 0,C 180,E1 16503.734,E2 16503.734} C_VEL
LIN {X 0,Y 349.193,Z 356.148,A -85,B 0,C 180,E1 16503.235,E2 16503.235} C_VEL
LIN {X 0,Y 347.501,Z 373.89,A -85,B 0,C 180,E1 16502.503,E2 16502.503} C_VEL
LIN {X 0,Y 345.317,Z 390.912,A -85,B 0,C 180,E1 16501.51,E2 16501.51} C_VEL
LIN {X 0,Y 342.793,Z 407.639,A -85,B 0,C 180,E1 16500.209,E2 16500.209} C_VEL
LIN {X 0,Y 339.961,Z 424.245,A -85,B 0,C 180,E1 16498.551,E2 16498.551} C_VEL
LIN {X 0,Y 337.264,Z 439.113,A -85,B 0,C 180,E1 16496.689,E2 16496.689} C_VEL
LIN {X 0,Y 334.679,Z 453.146,A -85,B 0,C 180,E1 16494.537,E2 16494.537} C_VEL
LIN {X 0,Y 332.371,Z 466.186,A -85,B 0,C 180,E1 16492.089,E2 16492.089} C_VEL
LIN {X 0,Y 330.554,Z 477.693,A -85,B 0,C 180,E1 16489.435,E2 16489.435} C_VEL
LIN {X 0,Y 329.286,Z 487.748,A -85,B 0,C 180,E1 16486.585,E2 16486.585} C_VEL
LIN {X 0,Y 328.645,Z 496.345,A -85,B 0,C 180,E1 16483.549,E2 16483.549} C_VEL
LIN {X 0,Y 328.564,Z 503.364,A -85,B 0,C 180,E1 16480.344,E2 16480.344} C_VEL
LIN {X 0,Y 328.905,Z 508.187,A -85,B 0,C 180,E1 16477.337,E2 16477.337} C_VEL
LIN {X 0,Y 329.378,Z 511.335,A -85,B 0,C 180,E1 16474.354,E2 16474.354} C_VEL
LIN {X 0,Y 329.721,Z 512.839,A -85,B 0,C 180,E1 16471.391,E2 16471.391} C_VEL
LIN {X 0,Y 329.735,Z 512.742,A -85,B 0,C 180,E1 16468.611,E2 16468.611} C_VEL
LIN {X 0,Y 329.448,Z 511.167,A -85,B 0,C 180,E1 16465.824,E2 16465.824} C_VEL
LIN {X 0,Y 328.996,Z 507.824,A -85,B 0,C 180,E1 16462.844,E2 16462.844} C_VEL
LIN {X 0,Y 328.653,Z 502.708,A -85,B 0,C 180,E1 16459.838,E2 16459.838} C_VEL
LIN {X 0,Y 328.678,Z 495.717,A -85,B 0,C 180,E1 16456.813,E2 16456.813} C_VEL
LIN {X 0,Y 329.164,Z 487.25,A -85,B 0,C 180,E1 16453.955,E2 16453.955} C_VEL
LIN {X 0,Y 330.238,Z 476.671,A -85,B 0,C 180,E1 16451.099,E2 16451.099} C_VEL
LIN {X 0,Y 331.709,Z 465.355,A -85,B 0,C 180,E1 16448.611,E2 16448.611} C_VEL
LIN {X 0,Y 333.649,Z 452.167,A -85,B 0,C 180,E1 16446.232,E2 16446.232} C_VEL
LIN {X 0,Y 335.811,Z 438.074,A -85,B 0,C 180,E1 16444.156,E2 16444.156} C_VEL
LIN {X 0,Y 338.09,Z 422.861,A -85,B 0,C 180,E1 16442.337,E2 16442.337} C_VEL
LIN {X 0,Y 340.415,Z 406.211,A -85,B 0,C 180,E1 16440.76,E2 16440.76} C_VEL
LIN {X 0,Y 342.448,Z 389.54,A -85,B 0,C 180,E1 16439.532,E2 16439.532} C_VEL
LIN {X 0,Y 344.279,Z 371.645,A -85,B 0,C 180,E1 16438.558,E2 16438.558} C_VEL
LIN {X 0,Y 345.584,Z 353.046,A -85,B 0,C 180,E1 16437.868,E2 16437.868} C_VEL
LIN {X 0,Y 346.481,Z 320.384,A -85,B 0,C 180,E1 16437.165,E2 16437.165} C_VEL
LIN {X 0,Y 350.199,Z 175.834,A -85,B 0,C 180,E1 16434.21,E2 16434.21} C_VEL
LIN {X 0,Y 349.623,Z 157.788,A -85,B 0,C 180,E1 16433.705,E2 16433.705} C_VEL
LIN {X 0,Y 352.142,Z 133.765,A -85,B 0,C 180,E1 16431.992,E2 16431.992} C_VEL
LIN {X 0,Y 343.157,Z 110.821,A -85,B 0,C 180,E1 16429.122,E2 16429.122} C_VEL
LIN {X 0,Y 334.538,Z 91.096,A -85,B 0,C 180,E1 16426.326,E2 16426.326} C_VEL
LIN {X 0,Y 330.132,Z 81.197,A -85,B 0,C 180,E1 16424.774,E2 16424.774} C_VEL
LIN {X 0,Y 330.052,Z 80.682,A -85,B 0,C 180,E1 16424.365,E2 16424.365} C_VEL
LIN {X 0,Y 330.054,Z 80.686,A -85,B 0,C 180,E1 16419.958,E2 16419.958} C_VEL
LIN {X 0,Y 330.041,Z 80.678,A -85,B 0,C 180,E1 16415.567,E2 16415.567} C_VEL
LIN {X 0,Y 330.046,Z 80.677,A -85,B 0,C 180,E1 16411.2,E2 16411.2} C_VEL
LIN {X 0,Y 330.053,Z 80.678,A -85,B 0,C 180,E1 16406.832,E2 16406.832} C_VEL
LIN {X 0,Y 330.055,Z 80.676,A -85,B 0,C 180,E1 16402.439,E2 16402.439} C_VEL
LIN {X 0,Y 330.034,Z 80.679,A -85,B 0,C 180,E1 16398,E2 16398} C_VEL
LIN {X 0,Y 330.035,Z 80.675,A -85,B 0,C 180,E1 16393.668,E2 16393.668} C_VEL
LIN {X 0,Y 330.043,Z 80.67,A -85,B 0,C 180,E1 16389.415,E2 16389.415} C_VEL
LIN {X 0,Y 330.049,Z 80.672,A -85,B 0,C 180,E1 16385.214,E2 16385.214} C_VEL
LIN {X 0,Y 330.046,Z 80.675,A -85,B 0,C 180,E1 16380.868,E2 16380.868} C_VEL
LIN {X 0,Y 330.028,Z 80.683,A -85,B 0,C 180,E1 16376.526,E2 16376.526} C_VEL
LIN {X 0,Y 330.026,Z 80.687,A -85,B 0,C 180,E1 16372.159,E2 16372.159} C_VEL
LIN {X 0,Y 330.041,Z 80.686,A -85,B 0,C 180,E1 16367.756,E2 16367.756} C_VEL
LIN {X 0,Y 330.051,Z 80.683,A -85,B 0,C 180,E1 16363.455,E2 16363.455} C_VEL
LIN {X 0,Y 330.028,Z 80.681,A -85,B 0,C 180,E1 16359.053,E2 16359.053} C_VEL
LIN {X 0,Y 330.016,Z 80.661,A -85,B 0,C 180,E1 16354.71,E2 16354.71} C_VEL
LIN {X 0,Y 330.019,Z 80.658,A -85,B 0,C 180,E1 16350.399,E2 16350.399} C_VEL
LIN {X 0,Y 330.038,Z 80.68,A -85,B 0,C 180,E1 16346.104,E2 16346.104} C_VEL
LIN {X 0,Y 330.036,Z 80.691,A -85,B 0,C 180,E1 16341.685,E2 16341.685} C_VEL
LIN {X 0,Y 330.072,Z 80.902,A -85,B 0,C 180,E1 16338.103,E2 16338.103} C_VEL
LIN {X 0,Y 331.964,Z 85.771,A -85,B 0,C 180,E1 16337.101,E2 16337.101} C_VEL
LIN {X 0,Y 337.906,Z 100.297,A -85,B 0,C 180,E1 16334.389,E2 16334.389} C_VEL
LIN {X 0,Y 343.344,Z 116.533,A -85,B 0,C 180,E1 16331.6,E2 16331.6} C_VEL
LIN {X 0,Y 346.184,Z 127.406,A -85,B 0,C 180,E1 16329.878,E2 16329.878} C_VEL
LIN {X 0,Y 344.775,Z 162.269,A -85,B 0,C 180,E1 16325.653,E2 16325.653} C_VEL
LIN {X 0,Y 343.52,Z 198.398,A -85,B 0,C 180,E1 16321.397,E2 16321.397} C_VEL
LIN {X 0,Y 343.359,Z 206.276,A -85,B 0,C 180,E1 16320.539,E2 16320.539} C_VEL
LIN {X 0,Y 344.003,Z 211.769,A -85,B 0,C 180,E1 16320.355,E2 16320.355} C_VEL
LIN {X 0,Y 341.789,Z 309.931,A -85,B 0,C 180,E1 16318.28,E2 16318.28} C_VEL
LIN {X 0,Y 341.708,Z 326.451,A -85,B 0,C 180,E1 16317.765,E2 16317.765} C_VEL
LIN {X 0,Y 341.157,Z 340.7,A -85,B 0,C 180,E1 16317.005,E2 16317.005} C_VEL
LIN {X 0,Y 340.209,Z 354.3,A -85,B 0,C 180,E1 16315.968,E2 16315.968} C_VEL
LIN {X 0,Y 338.989,Z 366.724,A -85,B 0,C 180,E1 16314.706,E2 16314.706} C_VEL
LIN {X 0,Y 337.448,Z 379.302,A -85,B 0,C 180,E1 16313.022,E2 16313.022} C_VEL
LIN {X 0,Y 335.821,Z 390.233,A -85,B 0,C 180,E1 16311.114,E2 16311.114} C_VEL
LIN {X 0,Y 334.288,Z 399.325,A -85,B 0,C 180,E1 16309.061,E2 16309.061} C_VEL
LIN {X 0,Y 332.972,Z 406.612,A -85,B 0,C 180,E1 16306.933,E2 16306.933} C_VEL
LIN {X 0,Y 331.786,Z 412.789,A -85,B 0,C 180,E1 16304.483,E2 16304.483} C_VEL
LIN {X 0,Y 330.928,Z 417.003,A -85,B 0,C 180,E1 16302.031,E2 16302.031} C_VEL
LIN {X 0,Y 330.364,Z 419.538,A -85,B 0,C 180,E1 16299.581,E2 16299.581} C_VEL
LIN {X 0,Y 330.031,Z 420.474,A -85,B 0,C 180,E1 16296.784,E2 16296.784} C_VEL
LIN {X 0,Y 329.994,Z 419.377,A -85,B 0,C 180,E1 16293.995,E2 16293.995} C_VEL
LIN {X 0,Y 330.221,Z 416.471,A -85,B 0,C 180,E1 16291.387,E2 16291.387} C_VEL
LIN {X 0,Y 330.684,Z 412.032,A -85,B 0,C 180,E1 16288.959,E2 16288.959} C_VEL
LIN {X 0,Y 331.412,Z 405.709,A -85,B 0,C 180,E1 16286.539,E2 16286.539} C_VEL
LIN {X 0,Y 332.345,Z 397.801,A -85,B 0,C 180,E1 16284.301,E2 16284.301} C_VEL
LIN {X 0,Y 333.431,Z 388.311,A -85,B 0,C 180,E1 16282.244,E2 16282.244} C_VEL
LIN {X 0,Y 334.545,Z 377.728,A -85,B 0,C 180,E1 16280.451,E2 16280.451} C_VEL
LIN {X 0,Y 335.633,Z 365.486,A -85,B 0,C 180,E1 16278.834,E2 16278.834} C_VEL
LIN {X 0,Y 336.611,Z 351.877,A -85,B 0,C 180,E1 16277.476,E2 16277.476} C_VEL
LIN {X 0,Y 337.332,Z 337.134,A -85,B 0,C 180,E1 16276.413,E2 16276.413} C_VEL
LIN {X 0,Y 337.628,Z 322.464,A -85,B 0,C 180,E1 16275.704,E2 16275.704} C_VEL
LIN {X 0,Y 337.598,Z 304.022,A -85,B 0,C 180,E1 16275.207,E2 16275.207} C_VEL
LIN {X 0,Y 338.258,Z 267.357,A -85,B 0,C 180,E1 16274.384,E2 16274.384} C_VEL
LIN {X 0,Y 338.951,Z 264.275,A -85,B 0,C 180,E1 16274.112,E2 16274.112} C_VEL
LIN {X 0,Y 339.777,Z 263.812,A -85,B 0,C 180,E1 16273.919,E2 16273.919} C_VEL
LIN {X 0,Y 341.785,Z 266.042,A -85,B 0,C 180,E1 16273.689,E2 16273.689} C_VEL
LIN {X 0,Y 343.52,Z 265.979,A -85,B 0,C 180,E1 16273.56,E2 16273.56} C_VEL
LIN {X 0,Y 342.459,Z 297.218,A -85,B 0,C 180,E1 16272.786,E2 16272.786} C_VEL
LIN {X 0,Y 340.944,Z 305.895,A -85,B 0,C 180,E1 16272.598,E2 16272.598} C_VEL
LIN {X 0,Y 335.37,Z 321.575,A -85,B 0,C 180,E1 16272.234,E2 16272.234} C_VEL
LIN {X 0,Y 333.557,Z 328.89,A -85,B 0,C 180,E1 16271.886,E2 16271.886} C_VEL
LIN {X 0,Y 333.317,Z 330.919,A -85,B 0,C 180,E1 16271.755,E2 16271.755} C_VEL
LIN {X 0,Y 331.994,Z 345.588,A -85,B 0,C 180,E1 16270.597,E2 16270.597} C_VEL
LIN {X 0,Y 330.339,Z 360.294,A -85,B 0,C 180,E1 16269.073,E2 16269.073} C_VEL
LIN {X 0,Y 328.712,Z 373.1,A -85,B 0,C 180,E1 16267.366,E2 16267.366} C_VEL
LIN {X 0,Y 327.105,Z 384.681,A -85,B 0,C 180,E1 16265.435,E2 16265.435} C_VEL
LIN {X 0,Y 325.516,Z 395.394,A -85,B 0,C 180,E1 16263.157,E2 16263.157} C_VEL
LIN {X 0,Y 324.265,Z 403.941,A -85,B 0,C 180,E1 16260.843,E2 16260.843} C_VEL
LIN {X 0,Y 323.242,Z 411.158,A -85,B 0,C 180,E1 16258.274,E2 16258.274} C_VEL
LIN {X 0,Y 322.572,Z 416.492,A -85,B 0,C 180,E1 16255.657,E2 16255.657} C_VEL
LIN {X 0,Y 322.202,Z 420.179,A -85,B 0,C 180,E1 16252.895,E2 16252.895} C_VEL
LIN {X 0,Y 322.142,Z 421.979,A -85,B 0,C 180,E1 16250.254,E2 16250.254} C_VEL
LIN {X 0,Y 322.408,Z 422.077,A -85,B 0,C 180,E1 16247.307,E2 16247.307} C_VEL
LIN {X 0,Y 322.992,Z 420.375,A -85,B 0,C 180,E1 16244.602,E2 16244.602} C_VEL
LIN {X 0,Y 323.982,Z 416.75,A -85,B 0,C 180,E1 16241.807,E2 16241.807} C_VEL
LIN {X 0,Y 325.301,Z 411.553,A -85,B 0,C 180,E1 16239.234,E2 16239.234} C_VEL
LIN {X 0,Y 327.127,Z 404.089,A -85,B 0,C 180,E1 16236.586,E2 16236.586} C_VEL
LIN {X 0,Y 329.126,Z 395.393,A -85,B 0,C 180,E1 16234.277,E2 16234.277} C_VEL
LIN {X 0,Y 331.428,Z 384.755,A -85,B 0,C 180,E1 16232.071,E2 16232.071} C_VEL
LIN {X 0,Y 333.854,Z 372.267,A -85,B 0,C 180,E1 16230.056,E2 16230.056} C_VEL
LIN {X 0,Y 336.058,Z 359.415,A -85,B 0,C 180,E1 16228.428,E2 16228.428} C_VEL
LIN {X 0,Y 338.24,Z 344.247,A -85,B 0,C 180,E1 16226.938,E2 16226.938} C_VEL
LIN {X 0,Y 339.978,Z 328.69,A -85,B 0,C 180,E1 16225.802,E2 16225.802} C_VEL
LIN {X 0,Y 341.267,Z 312.759,A -85,B 0,C 180,E1 16224.968,E2 16224.968} C_VEL
LIN {X 0,Y 342.337,Z 291.406,A -85,B 0,C 180,E1 16224.275,E2 16224.275} C_VEL
LIN {X 0,Y 346.454,Z 213.97,A -85,B 0,C 180,E1 16222.192,E2 16222.192} C_VEL
LIN {X 0,Y 341.856,Z 185.327,A -85,B 0,C 180,E1 16220.617,E2 16220.617} C_VEL
LIN {X 0,Y 339.361,Z 171.462,A -85,B 0,C 180,E1 16219.716,E2 16219.716} C_VEL
LIN {X 0,Y 344.408,Z 146.125,A -85,B 0,C 180,E1 16215.147,E2 16215.147} C_VEL
LIN {X 0,Y 341.67,Z 133.594,A -85,B 0,C 180,E1 16211.821,E2 16211.821} C_VEL
LIN {X 0,Y 338.619,Z 122.569,A -85,B 0,C 180,E1 16208.49,E2 16208.49} C_VEL
LIN {X 0,Y 335.525,Z 112.973,A -85,B 0,C 180,E1 16205.129,E2 16205.129} C_VEL
LIN {X 0,Y 332.531,Z 105.197,A -85,B 0,C 180,E1 16201.896,E2 16201.896} C_VEL
LIN {X 0,Y 330.361,Z 99.395,A -85,B 0,C 180,E1 16199.133,E2 16199.133} C_VEL
LIN {X 0,Y 328.158,Z 94.685,A -85,B 0,C 180,E1 16196.332,E2 16196.332} C_VEL
LIN {X 0,Y 326.497,Z 90.869,A -85,B 0,C 180,E1 16193.671,E2 16193.671} C_VEL
LIN {X 0,Y 324.295,Z 86.327,A -85,B 0,C 180,E1 16189.16,E2 16189.16} C_VEL
LIN {X 0,Y 322.821,Z 84.194,A -85,B 0,C 180,E1 16184.184,E2 16184.184} C_VEL
LIN {X 0,Y 322.798,Z 84.14,A -85,B 0,C 180,E1 16180.329,E2 16180.329} C_VEL
LIN {X 0,Y 324.329,Z 86.351,A -85,B 0,C 180,E1 16175.212,E2 16175.212} C_VEL
LIN {X 0,Y 325.18,Z 88.428,A -85,B 0,C 180,E1 16173.087,E2 16173.087} C_VEL
LIN {X 0,Y 327.299,Z 92.123,A -85,B 0,C 180,E1 16169.934,E2 16169.934} C_VEL
LIN {X 0,Y 329.514,Z 96.676,A -85,B 0,C 180,E1 16167.102,E2 16167.102} C_VEL
LIN {X 0,Y 331.716,Z 101.593,A -85,B 0,C 180,E1 16164.639,E2 16164.639} C_VEL
LIN {X 0,Y 333.854,Z 106.396,A -85,B 0,C 180,E1 16162.558,E2 16162.558} C_VEL
LIN {X 0,Y 336.509,Z 112.333,A -85,B 0,C 180,E1 16160.296,E2 16160.296} C_VEL
LIN {X 0,Y 340.488,Z 122.459,A -85,B 0,C 180,E1 16157.057,E2 16157.057} C_VEL
LIN {X 0,Y 344.474,Z 133.984,A -85,B 0,C 180,E1 16153.959,E2 16153.959} C_VEL
LIN {X 0,Y 348.183,Z 146.368,A -85,B 0,C 180,E1 16151.118,E2 16151.118} C_VEL
LIN {X 0,Y 348.738,Z 148.864,A -85,B 0,C 180,E1 16150.605,E2 16150.605} C_VEL
LIN {X 0,Y 345.576,Z 163.572,A -85,B 0,C 180,E1 16148.717,E2 16148.717} C_VEL
LIN {X 0,Y 348.462,Z 191.94,A -85,B 0,C 180,E1 16147.542,E2 16147.542} C_VEL
LIN {X 0,Y 343.46,Z 335.961,A -85,B 0,C 180,E1 16144.481,E2 16144.481} C_VEL
LIN {X 0,Y 342.48,Z 355.472,A -85,B 0,C 180,E1 16143.968,E2 16143.968} C_VEL
LIN {X 0,Y 340.652,Z 373.62,A -85,B 0,C 180,E1 16143.2,E2 16143.2} C_VEL
LIN {X 0,Y 338.452,Z 389.957,A -85,B 0,C 180,E1 16142.228,E2 16142.228} C_VEL
LIN {X 0,Y 335.792,Z 406.73,A -85,B 0,C 180,E1 16140.907,E2 16140.907} C_VEL
LIN {X 0,Y 332.819,Z 423.341,A -85,B 0,C 180,E1 16139.222,E2 16139.222} C_VEL
LIN {X 0,Y 329.971,Z 438.202,A -85,B 0,C 180,E1 16137.328,E2 16137.328} C_VEL
LIN {X 0,Y 327.224,Z 452.178,A -85,B 0,C 180,E1 16135.134,E2 16135.134} C_VEL
LIN {X 0,Y 324.759,Z 465.176,A -85,B 0,C 180,E1 16132.635,E2 16132.635} C_VEL
LIN {X 0,Y 322.802,Z 476.673,A -85,B 0,C 180,E1 16129.922,E2 16129.922} C_VEL
LIN {X 0,Y 321.415,Z 486.717,A -85,B 0,C 180,E1 16127.004,E2 16127.004} C_VEL
LIN {X 0,Y 320.689,Z 495.285,A -85,B 0,C 180,E1 16123.892,E2 16123.892} C_VEL
LIN {X 0,Y 320.567,Z 502.29,A -85,B 0,C 180,E1 16120.605,E2 16120.605} C_VEL
LIN {X 0,Y 320.911,Z 507.103,A -85,B 0,C 180,E1 16117.52,E2 16117.52} C_VEL
LIN {X 0,Y 321.413,Z 510.238,A -85,B 0,C 180,E1 16114.462,E2 16114.462} C_VEL
LIN {X 0,Y 321.779,Z 511.683,A -85,B 0,C 180,E1 16111.604,E2 16111.604} C_VEL
LIN {X 0,Y 321.822,Z 511.657,A -85,B 0,C 180,E1 16108.755,E2 16108.755} C_VEL
LIN {X 0,Y 321.525,Z 510.138,A -85,B 0,C 180,E1 16105.9,E2 16105.9} C_VEL
LIN {X 0,Y 321.045,Z 506.838,A -85,B 0,C 180,E1 16102.845,E2 16102.845} C_VEL
LIN {X 0,Y 320.681,Z 501.76,A -85,B 0,C 180,E1 16099.764,E2 16099.764} C_VEL
LIN {X 0,Y 320.708,Z 494.804,A -85,B 0,C 180,E1 16096.663,E2 16096.663} C_VEL
LIN {X 0,Y 321.223,Z 486.37,A -85,B 0,C 180,E1 16093.733,E2 16093.733} C_VEL
LIN {X 0,Y 322.354,Z 475.824,A -85,B 0,C 180,E1 16090.807,E2 16090.807} C_VEL
LIN {X 0,Y 323.898,Z 464.537,A -85,B 0,C 180,E1 16088.259,E2 16088.259} C_VEL
LIN {X 0,Y 325.927,Z 451.377,A -85,B 0,C 180,E1 16085.826,E2 16085.826} C_VEL
LIN {X 0,Y 328.185,Z 437.285,A -85,B 0,C 180,E1 16083.704,E2 16083.704} C_VEL
LIN {X 0,Y 330.557,Z 422.053,A -85,B 0,C 180,E1 16081.847,E2 16081.847} C_VEL
LIN {X 0,Y 332.886,Z 406.022,A -85,B 0,C 180,E1 16080.293,E2 16080.293} C_VEL
LIN {X 0,Y 335.03,Z 389.1,A -85,B 0,C 180,E1 16079.017,E2 16079.017} C_VEL
LIN {X 0,Y 336.915,Z 371.309,A -85,B 0,C 180,E1 16078.027,E2 16078.027} C_VEL
LIN {X 0,Y 338.281,Z 352.498,A -85,B 0,C 180,E1 16077.314,E2 16077.314} C_VEL
LIN {X 0,Y 339.209,Z 320.1,A -85,B 0,C 180,E1 16076.603,E2 16076.603} C_VEL
LIN {X 0,Y 343.103,Z 176.422,A -85,B 0,C 180,E1 16073.605,E2 16073.605} C_VEL
LIN {X 0,Y 342.515,Z 158.697,A -85,B 0,C 180,E1 16073.116,E2 16073.116} C_VEL
LIN {X 0,Y 344.955,Z 136.313,A -85,B 0,C 180,E1 16071.499,E2 16071.499} C_VEL
LIN {X 0,Y 336.036,Z 113.528,A -85,B 0,C 180,E1 16068.574,E2 16068.574} C_VEL
LIN {X 0,Y 327.124,Z 92.984,A -85,B 0,C 180,E1 16065.581,E2 16065.581} C_VEL
LIN {X 0,Y 322.276,Z 82.575,A -85,B 0,C 180,E1 16063.9,E2 16063.9} C_VEL
LIN {X 0,Y 322.109,Z 81.698,A -85,B 0,C 180,E1 16063.559,E2 16063.559} C_VEL
LIN {X 0,Y 322.111,Z 81.67,A -85,B 0,C 180,E1 16059.059,E2 16059.059} C_VEL
LIN {X 0,Y 322.114,Z 81.666,A -85,B 0,C 180,E1 16054.613,E2 16054.613} C_VEL
LIN {X 0,Y 322.117,Z 81.673,A -85,B 0,C 180,E1 16050.189,E2 16050.189} C_VEL
LIN {X 0,Y 322.1,Z 81.676,A -85,B 0,C 180,E1 16045.759,E2 16045.759} C_VEL
LIN {X 0,Y 322.108,Z 81.674,A -85,B 0,C 180,E1 16041.295,E2 16041.295} C_VEL
LIN {X 0,Y 322.114,Z 81.673,A -85,B 0,C 180,E1 16036.964,E2 16036.964} C_VEL
LIN {X 0,Y 322.111,Z 81.67,A -85,B 0,C 180,E1 16032.732,E2 16032.732} C_VEL
LIN {X 0,Y 322.098,Z 81.666,A -85,B 0,C 180,E1 16028.389,E2 16028.389} C_VEL
LIN {X 0,Y 322.09,Z 81.663,A -85,B 0,C 180,E1 16023.916,E2 16023.916} C_VEL
LIN {X 0,Y 322.113,Z 81.657,A -85,B 0,C 180,E1 16019.466,E2 16019.466} C_VEL
LIN {X 0,Y 322.102,Z 81.661,A -85,B 0,C 180,E1 16015.013,E2 16015.013} C_VEL
LIN {X 0,Y 322.088,Z 81.663,A -85,B 0,C 180,E1 16010.71,E2 16010.71} C_VEL
LIN {X 0,Y 322.082,Z 81.664,A -85,B 0,C 180,E1 16006.318,E2 16006.318} C_VEL
LIN {X 0,Y 322.097,Z 81.663,A -85,B 0,C 180,E1 16001.915,E2 16001.915} C_VEL
LIN {X 0,Y 322.111,Z 81.637,A -85,B 0,C 180,E1 15997.554,E2 15997.554} C_VEL
LIN {X 0,Y 322.084,Z 81.679,A -85,B 0,C 180,E1 15993.048,E2 15993.048} C_VEL
LIN {X 0,Y 322.077,Z 81.653,A -85,B 0,C 180,E1 15988.564,E2 15988.564} C_VEL
LIN {X 0,Y 322.087,Z 81.651,A -85,B 0,C 180,E1 15984.294,E2 15984.294} C_VEL
LIN {X 0,Y 322.108,Z 81.655,A -85,B 0,C 180,E1 15980.017,E2 15980.017} C_VEL
LIN {X 0,Y 322.121,Z 81.995,A -85,B 0,C 180,E1 15979.161,E2 15979.161} C_VEL
LIN {X 0,Y 328.224,Z 96.349,A -85,B 0,C 180,E1 15976.25,E2 15976.25} C_VEL
LIN {X 0,Y 334.108,Z 112.258,A -85,B 0,C 180,E1 15973.347,E2 15973.347} C_VEL
LIN {X 0,Y 338.681,Z 127.847,A -85,B 0,C 180,E1 15970.723,E2 15970.723} C_VEL
LIN {X 0,Y 339.173,Z 130.57,A -85,B 0,C 180,E1 15970.308,E2 15970.308} C_VEL
LIN {X 0,Y 337.746,Z 164.291,A -85,B 0,C 180,E1 15966.197,E2 15966.197} C_VEL
LIN {X 0,Y 336.417,Z 200.211,A -85,B 0,C 180,E1 15961.938,E2 15961.938} C_VEL
LIN {X 0,Y 336.234,Z 207.263,A -85,B 0,C 180,E1 15961.156,E2 15961.156} C_VEL
LIN {X 0,Y 336.895,Z 212.882,A -85,B 0,C 180,E1 15960.961,E2 15960.961} C_VEL
LIN {X 0,Y 334.574,Z 310.347,A -85,B 0,C 180,E1 15958.862,E2 15958.862} C_VEL
LIN {X 0,Y 334.485,Z 327.051,A -85,B 0,C 180,E1 15958.34,E2 15958.34} C_VEL
LIN {X 0,Y 333.926,Z 341.105,A -85,B 0,C 180,E1 15957.587,E2 15957.587} C_VEL
LIN {X 0,Y 332.982,Z 354.407,A -85,B 0,C 180,E1 15956.576,E2 15956.576} C_VEL
LIN {X 0,Y 331.66,Z 367.325,A -85,B 0,C 180,E1 15955.254,E2 15955.254} C_VEL
LIN {X 0,Y 330.108,Z 379.433,A -85,B 0,C 180,E1 15953.623,E2 15953.623} C_VEL
LIN {X 0,Y 328.487,Z 389.98,A -85,B 0,C 180,E1 15951.797,E2 15951.797} C_VEL
LIN {X 0,Y 326.815,Z 399.536,A -85,B 0,C 180,E1 15949.664,E2 15949.664} C_VEL
LIN {X 0,Y 325.304,Z 407.449,A -85,B 0,C 180,E1 15947.344,E2 15947.344} C_VEL
LIN {X 0,Y 324.029,Z 413.691,A -85,B 0,C 180,E1 15944.838,E2 15944.838} C_VEL
LIN {X 0,Y 323.101,Z 417.979,A -85,B 0,C 180,E1 15942.327,E2 15942.327} C_VEL
LIN {X 0,Y 322.454,Z 420.686,A -85,B 0,C 180,E1 15939.638,E2 15939.638} C_VEL
LIN {X 0,Y 322.118,Z 421.569,A -85,B 0,C 180,E1 15936.952,E2 15936.952} C_VEL
LIN {X 0,Y 322.06,Z 420.528,A -85,B 0,C 180,E1 15934.093,E2 15934.093} C_VEL
LIN {X 0,Y 322.288,Z 417.689,A -85,B 0,C 180,E1 15931.421,E2 15931.421} C_VEL
LIN {X 0,Y 322.764,Z 413.321,A -85,B 0,C 180,E1 15928.934,E2 15928.934} C_VEL
LIN {X 0,Y 323.516,Z 407.069,A -85,B 0,C 180,E1 15926.455,E2 15926.455} C_VEL
LIN {X 0,Y 324.571,Z 398.553,A -85,B 0,C 180,E1 15923.987,E2 15923.987} C_VEL
LIN {X 0,Y 325.717,Z 388.956,A -85,B 0,C 180,E1 15921.881,E2 15921.881} C_VEL
LIN {X 0,Y 326.83,Z 378.814,A -85,B 0,C 180,E1 15920.134,E2 15920.134} C_VEL
LIN {X 0,Y 327.978,Z 366.486,A -85,B 0,C 180,E1 15918.471,E2 15918.471} C_VEL
LIN {X 0,Y 328.995,Z 352.954,A -85,B 0,C 180,E1 15917.091,E2 15917.091} C_VEL
LIN {X 0,Y 329.725,Z 338.882,A -85,B 0,C 180,E1 15916.049,E2 15916.049} C_VEL
LIN {X 0,Y 330.062,Z 324.507,A -85,B 0,C 180,E1 15915.319,E2 15915.319} C_VEL
LIN {X 0,Y 330.056,Z 307.401,A -85,B 0,C 180,E1 15914.825,E2 15914.825} C_VEL
LIN {X 0,Y 330.301,Z 289.852,A -85,B 0,C 180,E1 15914.381,E2 15914.381} C_VEL
LIN {X 0,Y 331.041,Z 286.88,A -85,B 0,C 180,E1 15914.091,E2 15914.091} C_VEL
LIN {X 0,Y 331.849,Z 286.616,A -85,B 0,C 180,E1 15913.906,E2 15913.906} C_VEL
LIN {X 0,Y 333.688,Z 288.718,A -85,B 0,C 180,E1 15913.69,E2 15913.69} C_VEL
LIN {X 0,Y 335.407,Z 288.813,A -85,B 0,C 180,E1 15913.553,E2 15913.553} C_VEL
LIN {X 0,Y 334.701,Z 309.158,A -85,B 0,C 180,E1 15912.931,E2 15912.931} C_VEL
LIN {X 0,Y 333.745,Z 325.315,A -85,B 0,C 180,E1 15912.116,E2 15912.116} C_VEL
LIN {X 0,Y 333.317,Z 330.919,A -85,B 0,C 180,E1 15911.755,E2 15911.755} C_VEL
LIN {X 0,Y 331.8,Z 338.079,A -85,B 0,C 180,E1 15911.304,E2 15911.304} C_VEL
LIN {X 0,Y 325.566,Z 352.648,A -85,B 0,C 180,E1 15910.341,E2 15910.341} C_VEL
LIN {X 0,Y 323.013,Z 360.145,A -85,B 0,C 180,E1 15909.631,E2 15909.631} C_VEL
LIN {X 0,Y 322.695,Z 361.979,A -85,B 0,C 180,E1 15909.417,E2 15909.417} C_VEL
LIN {X 0,Y 320.913,Z 375.337,A -85,B 0,C 180,E1 15907.562,E2 15907.562} C_VEL
LIN {X 0,Y 319.246,Z 386.664,A -85,B 0,C 180,E1 15905.579,E2 15905.579} C_VEL
LIN {X 0,Y 317.625,Z 397.221,A -85,B 0,C 180,E1 15903.245,E2 15903.245} C_VEL
LIN {X 0,Y 316.335,Z 405.575,A -85,B 0,C 180,E1 15900.871,E2 15900.871} C_VEL
LIN {X 0,Y 315.289,Z 412.774,A -85,B 0,C 180,E1 15898.201,E2 15898.201} C_VEL
LIN {X 0,Y 314.591,Z 418.112,A -85,B 0,C 180,E1 15895.405,E2 15895.405} C_VEL
LIN {X 0,Y 314.253,Z 421.605,A -85,B 0,C 180,E1 15892.575,E2 15892.575} C_VEL
LIN {X 0,Y 314.24,Z 423.23,A -85,B 0,C 180,E1 15889.765,E2 15889.765} C_VEL
LIN {X 0,Y 314.564,Z 423.151,A -85,B 0,C 180,E1 15886.89,E2 15886.89} C_VEL
LIN {X 0,Y 315.28,Z 421.122,A -85,B 0,C 180,E1 15883.953,E2 15883.953} C_VEL
LIN {X 0,Y 316.356,Z 417.46,A -85,B 0,C 180,E1 15881.217,E2 15881.217} C_VEL
LIN {X 0,Y 317.899,Z 411.729,A -85,B 0,C 180,E1 15878.448,E2 15878.448} C_VEL
LIN {X 0,Y 319.772,Z 404.527,A -85,B 0,C 180,E1 15875.919,E2 15875.919} C_VEL
LIN {X 0,Y 322.121,Z 394.952,A -85,B 0,C 180,E1 15873.386,E2 15873.386} C_VEL
LIN {X 0,Y 324.423,Z 384.8,A -85,B 0,C 180,E1 15871.303,E2 15871.303} C_VEL
LIN {X 0,Y 326.968,Z 372.398,A -85,B 0,C 180,E1 15869.294,E2 15869.294} C_VEL
LIN {X 0,Y 329.222,Z 359.76,A -85,B 0,C 180,E1 15867.689,E2 15867.689} C_VEL
LIN {X 0,Y 331.44,Z 345.074,A -85,B 0,C 180,E1 15866.229,E2 15866.229} C_VEL
LIN {X 0,Y 333.314,Z 329.21,A -85,B 0,C 180,E1 15865.051,E2 15865.051} C_VEL
LIN {X 0,Y 334.676,Z 313.237,A -85,B 0,C 180,E1 15864.202,E2 15864.202} C_VEL
LIN {X 0,Y 335.808,Z 291.977,A -85,B 0,C 180,E1 15863.499,E2 15863.499} C_VEL
LIN {X 0,Y 340.098,Z 215.219,A -85,B 0,C 180,E1 15861.392,E2 15861.392} C_VEL
LIN {X 0,Y 335.675,Z 186.996,A -85,B 0,C 180,E1 15859.783,E2 15859.783} C_VEL
LIN {X 0,Y 332.837,Z 171.464,A -85,B 0,C 180,E1 15858.75,E2 15858.75} C_VEL
LIN {X 0,Y 337.509,Z 149.314,A -85,B 0,C 180,E1 15854.673,E2 15854.673} C_VEL
LIN {X 0,Y 334.944,Z 137.217,A -85,B 0,C 180,E1 15851.363,E2 15851.363} C_VEL
LIN {X 0,Y 332.052,Z 126.383,A -85,B 0,C 180,E1 15847.962,E2 15847.962} C_VEL
LIN {X 0,Y 329.197,Z 117.45,A -85,B 0,C 180,E1 15844.704,E2 15844.704} C_VEL
LIN {X 0,Y 326.356,Z 109.785,A -85,B 0,C 180,E1 15841.405,E2 15841.405} C_VEL
LIN {X 0,Y 324.018,Z 103.955,A -85,B 0,C 180,E1 15838.409,E2 15838.409} C_VEL
LIN {X 0,Y 322.578,Z 100.408,A -85,B 0,C 180,E1 15836.268,E2 15836.268} C_VEL
LIN {X 0,Y 320.841,Z 96.462,A -85,B 0,C 180,E1 15833.379,E2 15833.379} C_VEL
LIN {X 0,Y 318.999,Z 92.326,A -85,B 0,C 180,E1 15829.161,E2 15829.161} C_VEL
LIN {X 0,Y 317.624,Z 90.282,A -85,B 0,C 180,E1 15824.293,E2 15824.293} C_VEL
LIN {X 0,Y 317.602,Z 90.192,A -85,B 0,C 180,E1 15820.507,E2 15820.507} C_VEL
LIN {X 0,Y 319.093,Z 92.387,A -85,B 0,C 180,E1 15815.327,E2 15815.327} C_VEL
LIN {X 0,Y 319.895,Z 94.364,A -85,B 0,C 180,E1 15813.251,E2 15813.251} C_VEL
LIN {X 0,Y 321.96,Z 98.139,A -85,B 0,C 180,E1 15810.001,E2 15810.001} C_VEL
LIN {X 0,Y 324.116,Z 102.771,A -85,B 0,C 180,E1 15807.116,E2 15807.116} C_VEL
LIN {X 0,Y 326.144,Z 107.271,A -85,B 0,C 180,E1 15804.806,E2 15804.806} C_VEL
LIN {X 0,Y 329.115,Z 113.876,A -85,B 0,C 180,E1 15801.923,E2 15801.923} C_VEL
LIN {X 0,Y 333.169,Z 124.058,A -85,B 0,C 180,E1 15798.355,E2 15798.355} C_VEL
LIN {X 0,Y 337.124,Z 135.289,A -85,B 0,C 180,E1 15795.1,E2 15795.1} C_VEL
LIN {X 0,Y 340.85,Z 147.638,A -85,B 0,C 180,E1 15792.085,E2 15792.085} C_VEL
LIN {X 0,Y 341.925,Z 151.968,A -85,B 0,C 180,E1 15791.144,E2 15791.144} C_VEL
LIN {X 0,Y 339.278,Z 163.906,A -85,B 0,C 180,E1 15789.597,E2 15789.597} C_VEL
LIN {X 0,Y 342.108,Z 192.096,A -85,B 0,C 180,E1 15788.381,E2 15788.381} C_VEL
LIN {X 0,Y 337.073,Z 328.77,A -85,B 0,C 180,E1 15785.395,E2 15785.395} C_VEL
LIN {X 0,Y 336.045,Z 351.918,A -85,B 0,C 180,E1 15784.827,E2 15784.827} C_VEL
LIN {X 0,Y 334.289,Z 370.127,A -85,B 0,C 180,E1 15784.1,E2 15784.1} C_VEL
LIN {X 0,Y 331.935,Z 387.497,A -85,B 0,C 180,E1 15783.097,E2 15783.097} C_VEL
LIN {X 0,Y 329.191,Z 404.095,A -85,B 0,C 180,E1 15781.802,E2 15781.802} C_VEL
LIN {X 0,Y 326.179,Z 420.209,A -85,B 0,C 180,E1 15780.181,E2 15780.181} C_VEL
LIN {X 0,Y 322.977,Z 436.041,A -85,B 0,C 180,E1 15778.172,E2 15778.172} C_VEL
LIN {X 0,Y 320.028,Z 450.211,A -85,B 0,C 180,E1 15775.939,E2 15775.939} C_VEL
LIN {X 0,Y 317.348,Z 463.358,A -85,B 0,C 180,E1 15773.391,E2 15773.391} C_VEL
LIN {X 0,Y 315.189,Z 474.989,A -85,B 0,C 180,E1 15770.618,E2 15770.618} C_VEL
LIN {X 0,Y 313.616,Z 485.261,A -85,B 0,C 180,E1 15767.587,E2 15767.587} C_VEL
LIN {X 0,Y 312.757,Z 493.938,A -85,B 0,C 180,E1 15764.381,E2 15764.381} C_VEL
LIN {X 0,Y 312.563,Z 500.888,A -85,B 0,C 180,E1 15761.067,E2 15761.067} C_VEL
LIN {X 0,Y 312.915,Z 506.022,A -85,B 0,C 180,E1 15757.714,E2 15757.714} C_VEL
LIN {X 0,Y 313.451,Z 509.144,A -85,B 0,C 180,E1 15754.575,E2 15754.575} C_VEL
LIN {X 0,Y 313.85,Z 510.568,A -85,B 0,C 180,E1 15751.644,E2 15751.644} C_VEL
LIN {X 0,Y 313.909,Z 510.57,A -85,B 0,C 180,E1 15748.906,E2 15748.906} C_VEL
LIN {X 0,Y 313.604,Z 509.104,A -85,B 0,C 180,E1 15745.979,E2 15745.979} C_VEL
LIN {X 0,Y 313.094,Z 505.85,A -85,B 0,C 180,E1 15742.847,E2 15742.847} C_VEL
LIN {X 0,Y 312.707,Z 500.813,A -85,B 0,C 180,E1 15739.687,E2 15739.687} C_VEL
LIN {X 0,Y 312.741,Z 493.892,A -85,B 0,C 180,E1 15736.505,E2 15736.505} C_VEL
LIN {X 0,Y 313.281,Z 485.489,A -85,B 0,C 180,E1 15733.5,E2 15733.5} C_VEL
LIN {X 0,Y 314.383,Z 475.683,A -85,B 0,C 180,E1 15730.687,E2 15730.687} C_VEL
LIN {X 0,Y 316.098,Z 463.661,A -85,B 0,C 180,E1 15727.89,E2 15727.89} C_VEL
LIN {X 0,Y 318.223,Z 450.486,A -85,B 0,C 180,E1 15725.4,E2 15725.4} C_VEL
LIN {X 0,Y 320.578,Z 436.4,A -85,B 0,C 180,E1 15723.231,E2 15723.231} C_VEL
LIN {X 0,Y 323.049,Z 421.157,A -85,B 0,C 180,E1 15721.334,E2 15721.334} C_VEL
LIN {X 0,Y 325.466,Z 405.101,A -85,B 0,C 180,E1 15719.749,E2 15719.749} C_VEL
LIN {X 0,Y 327.638,Z 388.636,A -85,B 0,C 180,E1 15718.482,E2 15718.482} C_VEL
LIN {X 0,Y 329.581,Z 370.93,A -85,B 0,C 180,E1 15717.473,E2 15717.473} C_VEL
LIN {X 0,Y 330.999,Z 352.089,A -85,B 0,C 180,E1 15716.741,E2 15716.741} C_VEL
LIN {X 0,Y 331.946,Z 320.865,A -85,B 0,C 180,E1 15716.038,E2 15716.038} C_VEL
LIN {X 0,Y 336.041,Z 176.991,A -85,B 0,C 180,E1 15712.976,E2 15712.976} C_VEL
LIN {X 0,Y 335.491,Z 158.39,A -85,B 0,C 180,E1 15712.444,E2 15712.444} C_VEL
LIN {X 0,Y 337.769,Z 138.898,A -85,B 0,C 180,E1 15711.004,E2 15711.004} C_VEL
LIN {X 0,Y 329.135,Z 116.663,A -85,B 0,C 180,E1 15708.065,E2 15708.065} C_VEL
LIN {X 0,Y 320.469,Z 96.816,A -85,B 0,C 180,E1 15705.091,E2 15705.091} C_VEL
LIN {X 0,Y 315.23,Z 85.758,A -85,B 0,C 180,E1 15703.245,E2 15703.245} C_VEL
LIN {X 0,Y 314.221,Z 82.985,A -85,B 0,C 180,E1 15702.725,E2 15702.725} C_VEL
LIN {X 0,Y 314.171,Z 82.656,A -85,B 0,C 180,E1 15701.207,E2 15701.207} C_VEL
LIN {X 0,Y 314.174,Z 82.666,A -85,B 0,C 180,E1 15696.749,E2 15696.749} C_VEL
LIN {X 0,Y 314.176,Z 82.654,A -85,B 0,C 180,E1 15692.32,E2 15692.32} C_VEL
LIN {X 0,Y 314.164,Z 82.651,A -85,B 0,C 180,E1 15687.894,E2 15687.894} C_VEL
LIN {X 0,Y 314.164,Z 82.649,A -85,B 0,C 180,E1 15683.442,E2 15683.442} C_VEL
LIN {X 0,Y 314.175,Z 82.648,A -85,B 0,C 180,E1 15678.942,E2 15678.942} C_VEL
LIN {X 0,Y 314.173,Z 82.648,A -85,B 0,C 180,E1 15674.561,E2 15674.561} C_VEL
LIN {X 0,Y 314.154,Z 82.651,A -85,B 0,C 180,E1 15670.081,E2 15670.081} C_VEL
LIN {X 0,Y 314.159,Z 82.655,A -85,B 0,C 180,E1 15665.662,E2 15665.662} C_VEL
LIN {X 0,Y 314.177,Z 82.654,A -85,B 0,C 180,E1 15661.094,E2 15661.094} C_VEL
LIN {X 0,Y 314.156,Z 82.662,A -85,B 0,C 180,E1 15656.715,E2 15656.715} C_VEL
LIN {X 0,Y 314.149,Z 82.665,A -85,B 0,C 180,E1 15652.133,E2 15652.133} C_VEL
LIN {X 0,Y 314.165,Z 82.663,A -85,B 0,C 180,E1 15647.688,E2 15647.688} C_VEL
LIN {X 0,Y 314.167,Z 82.66,A -85,B 0,C 180,E1 15643.318,E2 15643.318} C_VEL
LIN {X 0,Y 314.144,Z 82.656,A -85,B 0,C 180,E1 15638.831,E2 15638.831} C_VEL
LIN {X 0,Y 314.149,Z 82.644,A -85,B 0,C 180,E1 15634.248,E2 15634.248} C_VEL
LIN {X 0,Y 314.176,Z 82.627,A -85,B 0,C 180,E1 15629.812,E2 15629.812} C_VEL
LIN {X 0,Y 314.148,Z 82.647,A -85,B 0,C 180,E1 15625.491,E2 15625.491} C_VEL
LIN {X 0,Y 314.132,Z 82.657,A -85,B 0,C 180,E1 15620.95,E2 15620.95} C_VEL
LIN {X 0,Y 314.215,Z 83.065,A -85,B 0,C 180,E1 15620.302,E2 15620.302} C_VEL
LIN {X 0,Y 320.692,Z 97.858,A -85,B 0,C 180,E1 15617.18,E2 15617.18} C_VEL
LIN {X 0,Y 326.551,Z 113.369,A -85,B 0,C 180,E1 15614.235,E2 15614.235} C_VEL
LIN {X 0,Y 331.276,Z 128.965,A -85,B 0,C 180,E1 15611.537,E2 15611.537} C_VEL
LIN {X 0,Y 332.318,Z 132.958,A -85,B 0,C 180,E1 15610.883,E2 15610.883} C_VEL
LIN {X 0,Y 330.666,Z 167.986,A -85,B 0,C 180,E1 15606.559,E2 15606.559} C_VEL
LIN {X 0,Y 329.26,Z 203.654,A -85,B 0,C 180,E1 15602.305,E2 15602.305} C_VEL
LIN {X 0,Y 329.189,Z 208.481,A -85,B 0,C 180,E1 15601.789,E2 15601.789} C_VEL
LIN {X 0,Y 329.822,Z 214.065,A -85,B 0,C 180,E1 15601.591,E2 15601.591} C_VEL
LIN {X 0,Y 327.396,Z 310.739,A -85,B 0,C 180,E1 15599.47,E2 15599.47} C_VEL
LIN {X 0,Y 327.303,Z 327.347,A -85,B 0,C 180,E1 15598.951,E2 15598.951} C_VEL
LIN {X 0,Y 326.733,Z 341.506,A -85,B 0,C 180,E1 15598.196,E2 15598.196} C_VEL
LIN {X 0,Y 325.794,Z 354.504,A -85,B 0,C 180,E1 15597.21,E2 15597.21} C_VEL
LIN {X 0,Y 324.361,Z 367.925,A -85,B 0,C 180,E1 15595.827,E2 15595.827} C_VEL
LIN {X 0,Y 322.789,Z 379.714,A -85,B 0,C 180,E1 15594.23,E2 15594.23} C_VEL
LIN {X 0,Y 321.206,Z 389.725,A -85,B 0,C 180,E1 15592.51,E2 15592.51} C_VEL
LIN {X 0,Y 319.405,Z 399.574,A -85,B 0,C 180,E1 15590.331,E2 15590.331} C_VEL
LIN {X 0,Y 317.763,Z 407.72,A -85,B 0,C 180,E1 15587.959,E2 15587.959} C_VEL
LIN {X 0,Y 316.459,Z 413.819,A -85,B 0,C 180,E1 15585.577,E2 15585.577} C_VEL
LIN {X 0,Y 315.407,Z 418.464,A -85,B 0,C 180,E1 15583.006,E2 15583.006} C_VEL
LIN {X 0,Y 314.616,Z 421.609,A -85,B 0,C 180,E1 15580.065,E2 15580.065} C_VEL
LIN {X 0,Y 314.204,Z 422.657,A -85,B 0,C 180,E1 15577.128,E2 15577.128} C_VEL
LIN {X 0,Y 314.123,Z 421.792,A -85,B 0,C 180,E1 15574.38,E2 15574.38} C_VEL
LIN {X 0,Y 314.31,Z 419.399,A -85,B 0,C 180,E1 15571.822,E2 15571.822} C_VEL
LIN {X 0,Y 314.802,Z 414.983,A -85,B 0,C 180,E1 15569.089,E2 15569.089} C_VEL
LIN {X 0,Y 315.552,Z 408.909,A -85,B 0,C 180,E1 15566.547,E2 15566.547} C_VEL
LIN {X 0,Y 316.534,Z 401.325,A -85,B 0,C 180,E1 15564.197,E2 15564.197} C_VEL
LIN {X 0,Y 317.692,Z 392.259,A -85,B 0,C 180,E1 15562.039,E2 15562.039} C_VEL
LIN {X 0,Y 319.005,Z 381.049,A -85,B 0,C 180,E1 15559.981,E2 15559.981} C_VEL
LIN {X 0,Y 320.257,Z 368.382,A -85,B 0,C 180,E1 15558.199,E2 15558.199} C_VEL
LIN {X 0,Y 321.322,Z 354.974,A -85,B 0,C 180,E1 15556.778,E2 15556.778} C_VEL
LIN {X 0,Y 322.103,Z 341.305,A -85,B 0,C 180,E1 15555.712,E2 15555.712} C_VEL
LIN {X 0,Y 322.51,Z 326.812,A -85,B 0,C 180,E1 15554.927,E2 15554.927} C_VEL
LIN {X 0,Y 322.681,Z 309.117,A -85,B 0,C 180,E1 15554.317,E2 15554.317} C_VEL
LIN {X 0,Y 323.464,Z 307.124,A -85,B 0,C 180,E1 15554.017,E2 15554.017} C_VEL
LIN {X 0,Y 324.291,Z 307.302,A -85,B 0,C 180,E1 15553.842,E2 15553.842} C_VEL
LIN {X 0,Y 326.2,Z 308.655,A -85,B 0,C 180,E1 15553.619,E2 15553.619} C_VEL
LIN {X 0,Y 327.414,Z 308.755,A -85,B 0,C 180,E1 15553.517,E2 15553.517} C_VEL
LIN {X 0,Y 326.461,Z 324.754,A -85,B 0,C 180,E1 15552.716,E2 15552.716} C_VEL
LIN {X 0,Y 325.166,Z 340.149,A -85,B 0,C 180,E1 15551.627,E2 15551.627} C_VEL
LIN {X 0,Y 323.449,Z 355.921,A -85,B 0,C 180,E1 15550.12,E2 15550.12} C_VEL
LIN {X 0,Y 322.695,Z 361.979,A -85,B 0,C 180,E1 15549.417,E2 15549.417} C_VEL
LIN {X 0,Y 320.946,Z 368.288,A -85,B 0,C 180,E1 15548.671,E2 15548.671} C_VEL
LIN {X 0,Y 314.776,Z 380.102,A -85,B 0,C 180,E1 15547.186,E2 15547.186} C_VEL
LIN {X 0,Y 311.928,Z 386.43,A -85,B 0,C 180,E1 15546.162,E2 15546.162} C_VEL
LIN {X 0,Y 311.381,Z 388.653,A -85,B 0,C 180,E1 15545.723,E2 15545.723} C_VEL
LIN {X 0,Y 309.763,Z 398.77,A -85,B 0,C 180,E1 15543.395,E2 15543.395} C_VEL
LIN {X 0,Y 308.327,Z 407.696,A -85,B 0,C 180,E1 15540.731,E2 15540.731} C_VEL
LIN {X 0,Y 307.325,Z 414.327,A -85,B 0,C 180,E1 15538.12,E2 15538.12} C_VEL
LIN {X 0,Y 306.625,Z 419.618,A -85,B 0,C 180,E1 15535.203,E2 15535.203} C_VEL
LIN {X 0,Y 306.311,Z 422.86,A -85,B 0,C 180,E1 15532.38,E2 15532.38} C_VEL
LIN {X 0,Y 306.333,Z 424.414,A -85,B 0,C 180,E1 15529.493,E2 15529.493} C_VEL
LIN {X 0,Y 306.694,Z 424.264,A -85,B 0,C 180,E1 15526.637,E2 15526.637} C_VEL
LIN {X 0,Y 307.495,Z 422.164,A -85,B 0,C 180,E1 15523.579,E2 15523.579} C_VEL
LIN {X 0,Y 308.695,Z 418.339,A -85,B 0,C 180,E1 15520.718,E2 15520.718} C_VEL
LIN {X 0,Y 310.385,Z 412.554,A -85,B 0,C 180,E1 15517.885,E2 15517.885} C_VEL
LIN {X 0,Y 312.405,Z 405.256,A -85,B 0,C 180,E1 15515.3,E2 15515.3} C_VEL
LIN {X 0,Y 314.716,Z 396.399,A -85,B 0,C 180,E1 15512.907,E2 15512.907} C_VEL
LIN {X 0,Y 317.234,Z 385.953,A -85,B 0,C 180,E1 15510.704,E2 15510.704} C_VEL
LIN {X 0,Y 320.004,Z 373.223,A -85,B 0,C 180,E1 15508.598,E2 15508.598} C_VEL
LIN {X 0,Y 322.463,Z 360.178,A -85,B 0,C 180,E1 15506.918,E2 15506.918} C_VEL
LIN {X 0,Y 324.82,Z 345.391,A -85,B 0,C 180,E1 15505.431,E2 15505.431} C_VEL
LIN {X 0,Y 326.78,Z 329.538,A -85,B 0,C 180,E1 15504.244,E2 15504.244} C_VEL
LIN {X 0,Y 328.197,Z 313.514,A -85,B 0,C 180,E1 15503.389,E2 15503.389} C_VEL
LIN {X 0,Y 329.397,Z 292.011,A -85,B 0,C 180,E1 15502.672,E2 15502.672} C_VEL
LIN {X 0,Y 333.819,Z 216.503,A -85,B 0,C 180,E1 15500.561,E2 15500.561} C_VEL
LIN {X 0,Y 329.596,Z 188.614,A -85,B 0,C 180,E1 15498.907,E2 15498.907} C_VEL
LIN {X 0,Y 326.487,Z 171.304,A -85,B 0,C 180,E1 15497.7,E2 15497.7} C_VEL
LIN {X 0,Y 330.653,Z 152.535,A -85,B 0,C 180,E1 15494.178,E2 15494.178} C_VEL
LIN {X 0,Y 328.274,Z 140.889,A -85,B 0,C 180,E1 15490.886,E2 15490.886} C_VEL
LIN {X 0,Y 325.631,Z 130.735,A -85,B 0,C 180,E1 15487.587,E2 15487.587} C_VEL
LIN {X 0,Y 322.867,Z 121.927,A -85,B 0,C 180,E1 15484.263,E2 15484.263} C_VEL
LIN {X 0,Y 320.101,Z 113.801,A -85,B 0,C 180,E1 15480.627,E2 15480.627} C_VEL
LIN {X 0,Y 317.87,Z 108.51,A -85,B 0,C 180,E1 15477.657,E2 15477.657} C_VEL
LIN {X 0,Y 316.762,Z 105.758,A -85,B 0,C 180,E1 15475.914,E2 15475.914} C_VEL
LIN {X 0,Y 315.331,Z 102.237,A -85,B 0,C 180,E1 15473.263,E2 15473.263} C_VEL
LIN {X 0,Y 313.612,Z 98.211,A -85,B 0,C 180,E1 15468.972,E2 15468.972} C_VEL
LIN {X 0,Y 312.381,Z 96.308,A -85,B 0,C 180,E1 15464.022,E2 15464.022} C_VEL
LIN {X 0,Y 312.449,Z 96.383,A -85,B 0,C 180,E1 15460.172,E2 15460.172} C_VEL
LIN {X 0,Y 314.126,Z 98.714,A -85,B 0,C 180,E1 15454.955,E2 15454.955} C_VEL
LIN {X 0,Y 316.536,Z 103.83,A -85,B 0,C 180,E1 15450.27,E2 15450.27} C_VEL
LIN {X 0,Y 318.688,Z 108.676,A -85,B 0,C 180,E1 15447.229,E2 15447.229} C_VEL
LIN {X 0,Y 320.576,Z 112.948,A -85,B 0,C 180,E1 15444.979,E2 15444.979} C_VEL
LIN {X 0,Y 323.294,Z 119.06,A -85,B 0,C 180,E1 15442.24,E2 15442.24} C_VEL
LIN {X 0,Y 327.123,Z 128.945,A -85,B 0,C 180,E1 15438.684,E2 15438.684} C_VEL
LIN {X 0,Y 330.812,Z 139.734,A -85,B 0,C 180,E1 15435.476,E2 15435.476} C_VEL
LIN {X 0,Y 334.402,Z 152.009,A -85,B 0,C 180,E1 15432.394,E2 15432.394} C_VEL
LIN {X 0,Y 335.141,Z 155.073,A -85,B 0,C 180,E1 15431.706,E2 15431.706} C_VEL
LIN {X 0,Y 333.069,Z 164.084,A -85,B 0,C 180,E1 15430.525,E2 15430.525} C_VEL
LIN {X 0,Y 335.818,Z 192.164,A -85,B 0,C 180,E1 15429.258,E2 15429.258} C_VEL
LIN {X 0,Y 334.771,Z 220.683,A -85,B 0,C 180,E1 15428.581,E2 15428.581} C_VEL
LIN {X 0,Y 329.764,Z 347.607,A -85,B 0,C 180,E1 15425.746,E2 15425.746} C_VEL
LIN {X 0,Y 328.072,Z 365.984,A -85,B 0,C 180,E1 15425.051,E2 15425.051} C_VEL
LIN {X 0,Y 325.663,Z 383.638,A -85,B 0,C 180,E1 15424.079,E2 15424.079} C_VEL
LIN {X 0,Y 322.869,Z 400.433,A -85,B 0,C 180,E1 15422.817,E2 15422.817} C_VEL
LIN {X 0,Y 319.806,Z 416.368,A -85,B 0,C 180,E1 15421.266,E2 15421.266} C_VEL
LIN {X 0,Y 316.496,Z 432.095,A -85,B 0,C 180,E1 15419.32,E2 15419.32} C_VEL
LIN {X 0,Y 313.267,Z 446.634,A -85,B 0,C 180,E1 15417.066,E2 15417.066} C_VEL
LIN {X 0,Y 310.369,Z 459.781,A -85,B 0,C 180,E1 15414.557,E2 15414.557} C_VEL
LIN {X 0,Y 307.897,Z 471.841,A -85,B 0,C 180,E1 15411.729,E2 15411.729} C_VEL
LIN {X 0,Y 306.059,Z 482.407,A -85,B 0,C 180,E1 15408.667,E2 15408.667} C_VEL
LIN {X 0,Y 304.94,Z 491.414,A -85,B 0,C 180,E1 15405.403,E2 15405.403} C_VEL
LIN {X 0,Y 304.567,Z 498.775,A -85,B 0,C 180,E1 15401.959,E2 15401.959} C_VEL
LIN {X 0,Y 304.796,Z 503.989,A -85,B 0,C 180,E1 15398.68,E2 15398.68} C_VEL
LIN {X 0,Y 305.342,Z 507.485,A -85,B 0,C 180,E1 15395.45,E2 15395.45} C_VEL
LIN {X 0,Y 305.831,Z 509.281,A -85,B 0,C 180,E1 15392.437,E2 15392.437} C_VEL
LIN {X 0,Y 306.013,Z 509.564,A -85,B 0,C 180,E1 15389.627,E2 15389.627} C_VEL
LIN {X 0,Y 305.764,Z 508.406,A -85,B 0,C 180,E1 15386.627,E2 15386.627} C_VEL
LIN {X 0,Y 305.275,Z 505.72,A -85,B 0,C 180,E1 15383.608,E2 15383.608} C_VEL
LIN {X 0,Y 304.806,Z 501.147,A -85,B 0,C 180,E1 15380.371,E2 15380.371} C_VEL
LIN {X 0,Y 304.719,Z 494.572,A -85,B 0,C 180,E1 15377.04,E2 15377.04} C_VEL
LIN {X 0,Y 305.193,Z 486.292,A -85,B 0,C 180,E1 15373.833,E2 15373.833} C_VEL
LIN {X 0,Y 306.319,Z 476.227,A -85,B 0,C 180,E1 15370.753,E2 15370.753} C_VEL
LIN {X 0,Y 308.034,Z 464.515,A -85,B 0,C 180,E1 15367.883,E2 15367.883} C_VEL
LIN {X 0,Y 310.1,Z 452.11,A -85,B 0,C 180,E1 15365.402,E2 15365.402} C_VEL
LIN {X 0,Y 312.567,Z 437.922,A -85,B 0,C 180,E1 15363.089,E2 15363.089} C_VEL
LIN {X 0,Y 315.164,Z 422.641,A -85,B 0,C 180,E1 15361.078,E2 15361.078} C_VEL
LIN {X 0,Y 317.644,Z 407.108,A -85,B 0,C 180,E1 15359.448,E2 15359.448} C_VEL
LIN {X 0,Y 319.91,Z 390.992,A -85,B 0,C 180,E1 15358.118,E2 15358.118} C_VEL
LIN {X 0,Y 322.025,Z 373.251,A -85,B 0,C 180,E1 15357.023,E2 15357.023} C_VEL
LIN {X 0,Y 323.566,Z 354.927,A -85,B 0,C 180,E1 15356.247,E2 15356.247} C_VEL
LIN {X 0,Y 324.386,Z 333.964,A -85,B 0,C 180,E1 15355.707,E2 15355.707} C_VEL
LIN {X 0,Y 329.059,Z 178.841,A -85,B 0,C 180,E1 15352.359,E2 15352.359} C_VEL
LIN {X 0,Y 328.517,Z 158.087,A -85,B 0,C 180,E1 15351.742,E2 15351.742} C_VEL
LIN {X 0,Y 330.549,Z 141.337,A -85,B 0,C 180,E1 15350.474,E2 15350.474} C_VEL
LIN {X 0,Y 321.832,Z 118.879,A -85,B 0,C 180,E1 15347.417,E2 15347.417} C_VEL
LIN {X 0,Y 313.001,Z 98.618,A -85,B 0,C 180,E1 15344.265,E2 15344.265} C_VEL
LIN {X 0,Y 307.594,Z 87.213,A -85,B 0,C 180,E1 15342.289,E2 15342.289} C_VEL
LIN {X 0,Y 306.293,Z 84.053,A -85,B 0,C 180,E1 15341.684,E2 15341.684} C_VEL
LIN {X 0,Y 306.235,Z 83.645,A -85,B 0,C 180,E1 15341.015,E2 15341.015} C_VEL
LIN {X 0,Y 306.236,Z 83.653,A -85,B 0,C 180,E1 15336.568,E2 15336.568} C_VEL
LIN {X 0,Y 306.234,Z 83.642,A -85,B 0,C 180,E1 15332.154,E2 15332.154} C_VEL
LIN {X 0,Y 306.223,Z 83.64,A -85,B 0,C 180,E1 15327.622,E2 15327.622} C_VEL
LIN {X 0,Y 306.237,Z 83.637,A -85,B 0,C 180,E1 15323.066,E2 15323.066} C_VEL
LIN {X 0,Y 306.233,Z 83.637,A -85,B 0,C 180,E1 15318.661,E2 15318.661} C_VEL
